//L2G2
arrfbLysGruppe[2]( 
	nZoneID:= 1, 
	bButtonZone1:= bTopButtonZone1,
	bBottomButtonZone1 := bBottomButtonZone1,
	//bButtonZone2:= bButtonZone2,
	fLuxOn:= fLuxOn, 
	fLuxDim:= fLuxDim, 
	tPIRDim:= tPIRDim, 
	tPIROff:= tPIROff, 
	fOffsetSec:= fOffsetSec, 
	bReInit:= , 
	stDaliSetup:= arrstDaliSetupGruppe[2], 
	ipCommunication_Prim:= P_DALI_Background.arrfbKL6821Communication[arrDALI_LINE_NUM_LIGHT[2]], 
	//ipCommunication_Sec:= P_DALI_Background.arrfbKL6821Communication[arrDALI_LINE_NUM_LIGHT[2]], 
	//ipCommunication_Supl:= P_DALI_Background.arrfbKL6821Communication[arrDALI_LINE_NUM_PENDANTS[2]], 
	fMinOutputPowerLevelRoom:= 15, 
	fMaxOutputPowerLevelRoom:= 100, 
	nCycleTimeInMS:= SH_Light.DALI_Param.nPlcTaskCycleTimeInMS*nDimCmdCycleTimeFactor,  //Used only for dim. Factor=2 makes dimming smooth 
	bRunTuning:= arrRunTuningGruppe[2], 
	bOccupiedRoom=> , 
	bError_Prim=> , 
	nError_Prim=> , 
	stTuneData:=arrstTuneDataGruppe[2] , 
	stPirSensorData:= stPirSensorData, 					//samme sensordata
	stLiveData:= arrstLiveDataGruppe[2]);
END_ACTION

ACTION A_ModbusComm:
//Manage data for modbus communication

//Manage data for read-only in PLC
stRoomDataPLC.bPirActive			:= stPirSensorData.bPrc;
stRoomDataPLC.uiActLuxLevel			:= TO_UINT(TRUNC(stPirSensorData.fBrightness));
stRoomDataPLC.uiActLightLevelPct	:= TO_UINT(TRUNC(arrfbLysGruppe[1].fbBallast.fActlLgtLvl_Prim));
		//stRoomDataPLC.uiActLightLevelPct	:= TO_UINT(TRUNC(fbLys.fbBallast.fActlLgtLvl_Prim)); //if only one group light control
stRoomDataPLC.uiBallastOnHours		:= uiBallastOnHours_MB; //The calculation for BallastOnHours is stored directly to the MB register below


//Assign data for read-only to MB registers
bPirActive_MB		:= stRoomDataPLC.bPirActive;
uiActLuxLevel_MB	:= stRoomDataPLC.uiActLuxLevel;

	//calculate BallastOnHours
	fbBallastOnHours(
		bEnableHourCount	:= bEnableHourCount,
		bPauseCount			:= arrfbLysGruppe[1].fbLightCtrl.bOffZone1,
		uiOnHours			:= uiBallastOnHours_MB,			//OnHours is updated here
		byOverflowCount		:= byOnHoursOverflowCount);


//Manage data for read/write for both PLC and MB registers
fbWriteSPLuxLevel(	nMaxValOut	:= uiMaxLuxLevel,
					nValIn1		:= uiSPLuxLevel_MB,		//nValIn1 takes priotity in case of download or restart
					nValIn2		:= stRoomDataPLC.uiSpLuxLevel,
					nValOut		=> uiLuxOn
				);


fbWritePirDelayTIme(	nMaxValOut	:= uiMaxPirOffMinutes,
						nValIn1		:= uiPirOffDelayTime_MB,		//nValIn1 takes priotity in case of download or restart
						nValIn2		:= stRoomDataPLC.uiPirOffDelayTime,
						nValOut		=> uiPirOffMinutes
					);
					

//Convert read/write modbus data to appropriate datatypes in PLC
fLuxOn	:= TO_REAL(uiLuxOn);			
tPIROff	:= TO_TIME(uiPirOffMinutes*udTimeScaling); //Time conversion defaults to ms

fLuxDim	:= TO_REAL(stRoomDataPLC.uiSpDimLuxLevel);			
tPIRDim	:= TO_TIME(stRoomDataPLC.uiPirDimDelayTime*udTimeScaling); //Time conversion defaults to ms
END_ACTION

ACTION A_Sensor:

fbSensor.ipCommunication := P_DALI_Background.arrfbKL6821Communication[Sensor_DALI_LINE_NUM];

//only 1 sensor
fbSensor(
	byShrtAdr:= bySensorAddr,
	bInitialize:= bInitialize, 
	DALI_LINE_NUM:= Sensor_DALI_LINE_NUM, 
 	//bCancelHoldTimerOccupancy:= bCancelHoldTimerOccupancy, 
	stSensorSetup := stDaliSensorSetup,
	bInitErr=> bInitErr, 
	bInitDone=> bInitDone,
	stPirSensorData:= stPirSensorData, 
	arrSensorScales:= arrSensorScales);


//several sensors
(*	
fbSensor(
	arrShrtAdr:= arrSensorAddr,
	bInitialize:= bInitialize, 
	DALI_LINE_NUM:= Sensor_DALI_LINE_NUM, 
 	//bCancelHoldTimerOccupancy:= bCancelHoldTimerOccupancy, 
	stSensorSetup := stDaliSensorSetup,
	arrInitErr=> arrInitErr, 
	arrInitDone=> arrInitDone,
	stPirSensorData:= stPirSensorData, 
	arrSensorScales:= arrSensorScales);
	*)
END_ACTION

END_PROGRAM

// ---- POUs/Alle_Rum/Rum_Med_DALI_Pir/Rum_4_213_Og_4_215_Foldedoer/P_Rum_4_215.TcPOU
PROGRAM P_Rum_4_215
VAR
(*Rummet består af to lysgrupper - L1G7 og L2G7 - på to forskellige linjer
Begge grupper afhænger af samme PIR-input - pir-adr. 5 og 8 - på DALI-linje 2.
Derfor oprettes to adskilte reguleringer med samme PV.
Yderligere logik for knapfunktion og pirsignaler håndteres i program for foldedør.
*)

	arrfbLysGruppe			: ARRAY [1..2] OF SH_Light.FB_Light_Type_A;
	arrstDaliSetupGruppe	: ARRAY [1..2] OF SH_Light.ST_DALI_RoomSetup := 
	
													[(	byShrtAdr_Prim := 18, 
														byGrpAdr_Prim := 7, 
														eMod_Prim := E_DALIAddressType.Group, 
														//byShrtAdr_Sec := 1, 
														//byGrpAdr_Sec := 1, 
														//eMod_Sec := E_DALIAddressType.Short, 
														//byShrtAdr_Supl := 1,
														//byGrpAdr_Supl := 1,
														//eMod_Supl := E_DALIADDRESSTYPE.Group,
														DALI_LINE_NUM_PRIM := arrDALI_LINE_NUM_LIGHT[1], 
														DALI_LINE_NUM_SEC := 0, //0 = ingen zonestyring/vinduerække
														DALI_LINE_NUM_SUPL := arrDALI_LINE_NUM_PENDANTS[1]),
														
													(	byShrtAdr_Prim := 13, 
														byGrpAdr_Prim := 7, 
														eMod_Prim := E_DALIAddressType.Group,
														//byShrtAdr_Sec := 1, 
														//byGrpAdr_Sec := 1, 
														//eMod_Sec := E_DALIAddressType.Short, 
														//byShrtAdr_Supl := 1,
														//byGrpAdr_Supl := 1,
														//eMod_Supl := E_DALIAddressType.Group, 
														DALI_LINE_NUM_PRIM := arrDALI_LINE_NUM_LIGHT[2], 
														DALI_LINE_NUM_SEC := 0, 
														DALI_LINE_NUM_SUPL := arrDALI_LINE_NUM_PENDANTS[2])];
														
	arrstLiveDataGruppe		: ARRAY [1..2] OF SH_Light.ST_LiveData;
	
	arrRunTuningGruppe: ARRAY[1..2] OF BOOL;
	
	bTopButtonZone1				: BOOL;
	bTopButtonZone1_Visu		: BOOL;
	bBottomButtonZone1			: BOOL;
	bBottomButtonZone1_Visu	: BOOL;
	bButtonZone2					: BOOL;
	bNeighborRoomsPir			: BOOL;
	fLuxOn								: REAL; 
	fLuxDim							: REAL;
	tPIRDim							: TIME;
	tPIROff							: TIME;
	fOffsetSec						: REAL := 20;
 

// Sensor Settings
	//fbSensor					: SH_Light.FB_NIKO_P46xx_1Pcs;
	fbSensor						: SH_Light.FB_NIKO_P46xx_2Pcs;
	//bySensorAddr				: BYTE := 1;
	arrSensorAddr				: ARRAY[1..2] OF BYTE := [5,8];
	bInitialize						: BOOL := TRUE;
	stDaliSensorSetup			: ST_DALI_NIKOP46SetupData;
	//bInitErr							: BOOL;
	//bInitDone						: BOOL;
	arrInitErr						: ARRAY [1..2] OF BOOL;
	arrInitDone					: ARRAY [1..2] OF BOOL;
	arrSensorScales				: ARRAY [1..10] OF SH_Light.ST_DALI_SensorScaleMode :=
																					[	(fMeassureMaxSensor := rMeassure_Zone5, fReadMaxSensor := rRead_Zone5),																		
																						(fMeassureMaxSensor := rMeassure_Zone5, fReadMaxSensor := rRead_Zone5),	
																						8(())];
																																			
	bCancelHoldTimerOccupancy	: BOOL;
(*	eEventPriorityOccupancy		: E_DALIEventPriority := E_DALIEVENTPRIORITY.Middle;
	nHoldTimerOccupancy			: WORD := 5; // Value in s. 	
	nReportTimerOccupancy		: BYTE := 120; // Value in s, Preset manufacturer value
	nDeadtimeTimerOccupancy		: WORD := 100; // Value in ms, Predefined Value of DALI Standard
	bCancelHoldTimerOccupancy	: BOOL;
	nSensitivityOccupancy		: BYTE:= 3; //setting Sensivity (0..4) 0 (Off), 1 (Min), 2(Low), 3(High) and 4 (Max)

	bEnableLuxEvent				: BOOL;
	eEventPriorityBrightness	: E_DALIEventPriority := E_DALIEVENTPRIORITY.Middle;
	nDeadtimeTimerBrightness	: WORD := 1500; // Value in ms, Predefined Value of DALI Standard
	nHysteresisBrightness		: BYTE := 2; // Value in %
	nHysteresisMinBrightness	: BYTE := 10; // Absolute Value, depending on the manufacturer specific resolution
	nReportTimerBrightness		: BYTE := 120; // Value in s, Preset manufacturer value
*)


//ModbusComm setup
	
	fbWriteSPLuxLevel				: SH_Light.FB_TwoVal_SelectOne_RTrigChange;
	fbWritePirDelayTIme			: SH_Light.FB_TwoVal_SelectOne_RTrigChange;
	stRoomDataPLC					: SH_Light.ST_RoomDataPLC	:=	(	uiPirOffDelayTime	:= 30,
																										uiSpLuxLevel			:= 500,
																										uiPirDimDelayTime	:= 15,
																										uiSpDimLuxLevel		:= 200);
																
	fbBallastOnHours					: SH_Light.FB_CountOnHours;
	bEnableHourCount				: BOOL := TRUE;
	
	//Non-persistent modbus data
	bPirActive_MB					AT%MX144.0	: BOOL;				//bPirLys i gammel kode
	uiActLuxLevel_MB			AT%MB148		: UINT;				//intHMIAktueltLux i gammel kode
	uiActLightLevelPct_MB	AT%MB156		: UINT;				//intDALI_Gruppe1_Lysniveau i gammel kode
	
	//For Conversion
	uiPirOffMinutes						: UINT;
	udTimeScaling						: UDINT := 60000;
	uiLuxOn								: UINT;
	
	//max values checks
	uiMaxLuxLevel						: UINT := 1023;
	uiMaxPirOffMinutes					: UINT := 180;
	
END_VAR

VAR CONSTANT
	Sensor_DALI_LINE_NUM					: BYTE := 2;
	arrDALI_LINE_NUM_LIGHT				: ARRAY[1..2] OF BYTE := [1,2]; //korrekt rækkefølge nødvendig //rækkefølge og linje 
	arrDALI_LINE_NUM_PENDANTS	: ARRAY[1..2] OF BYTE := [0,0]; //korrekt rækkefølge nødvendig. 0 = ingen pendler
END_VAR

VAR PERSISTENT
	stPirSensorData										: SH_Light.ST_DALI_Sensor;
	arrstTuneDataGruppe								: ARRAY [1..2] OF SH_Light.ST_TuneData_EX;

	uiPirOffDelayTime_MB		AT%MB146	    : UINT;				//intHMI_Pir_SetValue i gammel kode
	uiSPLuxLevel_MB		    AT%MB152    	: UINT;				//intHMI_Lux_SetValue i gammel kode
	uiBallastOnHours_MB	    AT%MB158	    : UINT;				//dintHMILysbraendtimer1 i gammel kode
	byOnHoursOverflowCount			   				: BYTE;
END_VAR

A_Buttons();
A_LightCtrl();
A_ModbusComm();
A_Sensor();

ACTION A_Buttons:
//Logik for knapper håndteres i P_Foldedoer_4_213

bTopButtonZone1		:= P_Foldedoer_4_213.arrTopButtonZone1Comb[2] OR bTopButtonZone1_Visu;
bBottomButtonZone1	:= P_Foldedoer_4_213.arrBottomButtonZone1Comb[2] OR bBottomButtonZone1_Visu;
END_ACTION

ACTION A_LightCtrl:
  
//gruppe L1G1
arrfbLysGruppe[1]( 
	nZoneID:= 1, 
	bButtonZone1:= bTopButtonZone1,
	bBottomButtonZone1 := bBottomButtonZone1,
	//bButtonZone2:= bButtonZone2,
	fLuxOn:= fLuxOn, 
	fLuxDim:= fLuxDim, 
	tPIRDim:= tPIRDim, 
	tPIROff:= tPIROff, 
	fOffsetSec:= fOffsetSec, 
	bReInit:= , 
	stDaliSetup:= arrstDaliSetupGruppe[1], 
	ipCommunication_Prim:= P_DALI_Background.arrfbKL6821Communication[arrDALI_LINE_NUM_LIGHT[1]], 
	//ipCommunication_Sec:= P_DALI_Background.arrfbKL6821Communication[arrDALI_LINE_NUM_LIGHT[1]], 
	//ipCommunication_Supl:= P_DALI_Background.arrfbKL6821Communication[arrDALI_LINE_NUM_PENDANTS[1]], 
	fMinOutputPowerLevelRoom:= 15, 
	fMaxOutputPowerLevelRoom:= 100, 
	nCycleTimeInMS:= SH_Light.DALI_Param.nPlcTaskCycleTimeInMS*nDimCmdCycleTimeFactor,   //Used only for dim. Factor=2 makes dimming smooth
	bRunTuning:= arrRunTuningGruppe[1], 
	bOccupiedRoom=> , 
	bError_Prim=> , 
	nError_Prim=> , 
	stTuneData:=arrstTuneDataGruppe[1] , 
	stPirSensorData:=  P_Foldedoer_4_213.arrstPirSensorDataComb[2], 					//samme sensordata
	stLiveData:= arrstLiveDataGruppe[1]);

//gruppe 15	
arrfbLysGruppe[2]( 
	nZoneID:= 1, 
	bButtonZone1:= bTopButtonZone1,
	bBottomButtonZone1 := bBottomButtonZone1,
	//bButtonZone2:= bButtonZone2,
	fLuxOn:= fLuxOn, 
	fLuxDim:= fLuxDim, 
	tPIRDim:= tPIRDim, 
	tPIROff:= tPIROff, 
	fOffsetSec:= fOffsetSec, 
	bReInit:= , 
	stDaliSetup:= arrstDaliSetupGruppe[2], 
	ipCommunication_Prim:= P_DALI_Background.arrfbKL6821Communication[arrDALI_LINE_NUM_LIGHT[2]], 
	//ipCommunication_Sec:= P_DALI_Background.arrfbKL6821Communication[arrDALI_LINE_NUM_LIGHT[2]], 
	//ipCommunication_Supl:= P_DALI_Background.arrfbKL6821Communication[arrDALI_LINE_NUM_PENDANTS[2]], 
	fMinOutputPowerLevelRoom:= 15, 
	fMaxOutputPowerLevelRoom:= 100, 
	nCycleTimeInMS:= SH_Light.DALI_Param.nPlcTaskCycleTimeInMS*nDimCmdCycleTimeFactor,  //Used only for dim. Factor=2 makes dimming smooth
	bRunTuning:= arrRunTuningGruppe[2], 
	bOccupiedRoom=> , 
	bError_Prim=> , 
	nError_Prim=> , 
	stTuneData:=arrstTuneDataGruppe[2] , 
	stPirSensorData:=  P_Foldedoer_4_213.arrstPirSensorDataComb[2], 					//samme sensordata
	stLiveData:= arrstLiveDataGruppe[2]);
END_ACTION

ACTION A_ModbusComm:
//Manage data for modbus communication

//Manage data for read-only in PLC
stRoomDataPLC.bPirActive			:= stPirSensorData.bPrc;
stRoomDataPLC.uiActLuxLevel			:= TO_UINT(TRUNC(stPirSensorData.fBrightness));
stRoomDataPLC.uiActLightLevelPct	:= TO_UINT(TRUNC(arrfbLysGruppe[1].fbBallast.fActlLgtLvl_Prim));
		//stRoomDataPLC.uiActLightLevelPct	:= TO_UINT(TRUNC(fbLys.fbBallast.fActlLgtLvl_Prim)); //if only one group light control
stRoomDataPLC.uiBallastOnHours		:= uiBallastOnHours_MB; //The calculation for BallastOnHours is stored directly to the MB register below


//Assign data for read-only to MB registers
bPirActive_MB		:= stRoomDataPLC.bPirActive;
uiActLuxLevel_MB	:= stRoomDataPLC.uiActLuxLevel;

	//calculate BallastOnHours
	fbBallastOnHours(
		bEnableHourCount	:= bEnableHourCount,
		bPauseCount			:= arrfbLysGruppe[1].fbLightCtrl.bOffZone1,
		uiOnHours			:= uiBallastOnHours_MB,			//OnHours is updated here
		byOverflowCount		:= byOnHoursOverflowCount);


//Manage data for read/write for both PLC and MB registers
fbWriteSPLuxLevel(	nMaxValOut	:= uiMaxLuxLevel,
					nValIn1		:= uiSPLuxLevel_MB,		//nValIn1 takes priotity in case of download or restart
					nValIn2		:= stRoomDataPLC.uiSpLuxLevel,
					nValOut		=> uiLuxOn
				);


fbWritePirDelayTIme(	nMaxValOut	:= uiMaxPirOffMinutes,
						nValIn1		:= uiPirOffDelayTime_MB,		//nValIn1 takes priotity in case of download or restart
						nValIn2		:= stRoomDataPLC.uiPirOffDelayTime,
						nValOut		=> uiPirOffMinutes
					);
					

//Convert read/write modbus data to appropriate datatypes in PLC
fLuxOn	:= TO_REAL(uiLuxOn);			
tPIROff	:= TO_TIME(uiPirOffMinutes*udTimeScaling); //Time conversion defaults to ms

fLuxDim	:= TO_REAL(stRoomDataPLC.uiSpDimLuxLevel);			
tPIRDim	:= TO_TIME(stRoomDataPLC.uiPirDimDelayTime*udTimeScaling); //Time conversion defaults to ms
END_ACTION

ACTION A_Sensor:

fbSensor.ipCommunication := P_DALI_Background.arrfbKL6821Communication[Sensor_DALI_LINE_NUM];

//only 1 sensor
(*
fbSensor(
	byShrtAdr:= bySensorAddr,
	bInitialize:= bInitialize, 
	DALI_LINE_NUM:= Sensor_DALI_LINE_NUM, 
 	//bCancelHoldTimerOccupancy:= bCancelHoldTimerOccupancy, 
	stSensorSetup := stDaliSensorSetup,
	bInitErr=> bInitErr, 
	bInitDone=> bInitDone,
	stPirSensorData:= stPirSensorData, 
	arrSensorScales:= arrSensorScales);
*)

//several sensors
fbSensor(
	arrShrtAdr:= arrSensorAddr,
	bInitialize:= bInitialize, 
	DALI_LINE_NUM:= Sensor_DALI_LINE_NUM, 
 	//bCancelHoldTimerOccupancy:= bCancelHoldTimerOccupancy, 
	stSensorSetup := stDaliSensorSetup,
	arrInitErr=> arrInitErr, 
	arrInitDone=> arrInitDone,
	stPirSensorData := P_Foldedoer_4_213.arrstPirSensorData[2], 
	arrSensorScales:= arrSensorScales);
	
	stPirSensorData := P_Foldedoer_4_213.arrstPirSensorData[2]; //For at holde samme navngivning i A_ModbusComm
END_ACTION

END_PROGRAM

// ---- POUs/Alle_Rum/Gange/Gang_4_210A/P_Gang_4_210A.TcPOU
PROGRAM P_Gang_4_210A
VAR
//Light

	fbLys			: SH_Light.FB_Light_Type_B;
	
	stDaliSetup	: SH_Light.ST_DALI_RoomSetup := (
														byShrtAdr_Prim	:= 56, 
														byGrpAdr_Prim		:= 1, 
														eMod_Prim			:= E_DALIAddressType.Group, 
														//byShrtAdr_Sec	:= 1, 
														//byGrpAdr_Sec	:= 1, 
														//eMod_Sec			:= E_DALIAddressType.Short, 
														//byShrtAdr_Supl		:= 1,
														//byGrpAdr_Supl		:= 1,
														//eMod_Supl			:= Tc3_DALI.E_DALIAddressType.Short, 
														DALI_LINE_NUM_PRIM := DALI_LINE_NUM_LIGHT, 
														DALI_LINE_NUM_SEC := 0, 
														DALI_LINE_NUM_SUPL := DALI_LINE_NUM_PENDANT);
														
	stLiveData						: SH_Light.ST_LiveData;
	bRunTuning						: BOOL;
	
	bTopButtonZone1				: BOOL;
	bTopButtonZone1_Visu		: BOOL;
	bBottomButtonZone1			: BOOL;
	bBottomButtonZone1_Visu	: BOOL;
	bButtonZone2					: BOOL;
	fLuxOn								: REAL;
	fLuxDim							: REAL;
	tPIRDim							: TIME;
	tPIROff							: TIME;
	fOffsetSec						: REAL := 20;
	bOccupiedRoom				: BOOL;
	
// Sensor Settings
	fbSensor							: SH_Light.FB_NIKO_P46xx_1Pcs;
	//fbSensor							: SH_Light.FB_NIKO_P46xx_2Pcs;
	bySensorAddr					: BYTE := 63;
	//arrSensorAddr					: ARRAY[1..2] OF BYTE := [3,4];
	bInitialize							: BOOL := TRUE;
	stDaliSensorSetup				: ST_DALI_NIKOP46SetupData;
	bInitErr								: BOOL;
	bInitDone							: BOOL;
	//arrInitErr							: ARRAY [1..2] OF BOOL;
	//arrInitDone						: ARRAY [1..2] OF BOOL;
	arrSensorScales					: ARRAY [1..10] OF SH_Light.ST_DALI_SensorScaleMode :=
																						[	(fMeassureMaxSensor := rMeassure_Zone10, fReadMaxSensor := rRead_Zone10),
																							9(())];
	bCancelHoldTimerOccupancy	: BOOL;
(*	eEventPriorityOccupancy		: E_DALIEventPriority := E_DALIEVENTPRIORITY.Middle;
	nHoldTimerOccupancy			: WORD := 5; // Value in s. 	
	nReportTimerOccupancy		: BYTE := 120; // Value in s, Preset manufacturer value
	nDeadtimeTimerOccupancy		: WORD := 100; // Value in ms, Predefined Value of DALI Standard
	bCancelHoldTimerOccupancy	: BOOL;
	nSensitivityOccupancy		: BYTE:= 3; //setting Sensivity (0..4) 0 (Off), 1 (Min), 2(Low), 3(High) and 4 (Max)

	bEnableLuxEvent				: BOOL;
	eEventPriorityBrightness	: E_DALIEventPriority := E_DALIEVENTPRIORITY.Middle;
	nDeadtimeTimerBrightness	: WORD := 1500; // Value in ms, Predefined Value of DALI Standard
	nHysteresisBrightness		: BYTE := 2; // Value in %
	nHysteresisMinBrightness	: BYTE := 10; // Absolute Value, depending on the manufacturer specific resolution
	nReportTimerBrightness		: BYTE := 120; // Value in s, Preset manufacturer value
*)

//ModbusComm setup
	
	fbWriteSPLuxLevel				: SH_Light.FB_TwoVal_SelectOne_RTrigChange;
	fbWritePirDelayTIme			: SH_Light.FB_TwoVal_SelectOne_RTrigChange;
	stRoomDataPLC					: SH_Light.ST_RoomDataPLC	:=	(	uiPirOffDelayTime	:= 30,
																										uiSpLuxLevel			:= 500,
																										uiPirDimDelayTime	:= 15,
																										uiSpDimLuxLevel		:= 200);
																
	fbBallastOnHours					: SH_Light.FB_CountOnHours;
	bEnableHourCount				: BOOL := TRUE;
	
	//Non-persistent modbus data
	bPirActive_MB					AT%MX200.0	: BOOL;				//bPirLys i gammel kode
	uiActLuxLevel_MB			AT%MB204		: UINT;				//intHMIAktueltLux i gammel kode
	uiActLightLevelPct_MB	AT%MB208		: UINT;				//intDALI_Gruppe1_Lysniveau i gammel kode
	
	//For Conversion
	uiPirOffMinutes						: UINT;
	udTimeScaling						: UDINT := 60000;
	uiLuxOn								: UINT;
	
	//max values checks
	uiMaxLuxLevel						: UINT := 1023;
	uiMaxPirOffMinutes				: UINT := 180;

END_VAR

VAR CONSTANT
	Sensor_DALI_LINE_NUM: BYTE := 3;
	DALI_LINE_NUM_LIGHT: BYTE := 3;
	DALI_LINE_NUM_PENDANT: BYTE :=0;
END_VAR
VAR PERSISTENT
	stPirSensorData: SH_Light.ST_DALI_Sensor;
	stTuneData: SH_Light.ST_TuneData_EX;
	
	uiPirOffDelayTime_MB		AT%MB202	    : UINT;				//intHMI_Pir_SetValue i gammel kode
	uiSPLuxLevel_MB		    AT%MB206    	: UINT;				//intHMI_Lux_SetValue i gammel kode
	uiBallastOnHours_MB	    AT%MB210	    : UINT;				//dintHMILysbraendtimer1 i gammel kode
	byOnHoursOverflowCount			   				: BYTE;
END_VAR

A_Buttons();
A_LightCtrl();
A_ModbusComm();
A_Sensor();

ACTION A_Buttons:
bTopButtonZone1		:= 	bTopButtonZone1_Visu;
bBottomButtonZone1	:= 	bBottomButtonZone1_Visu;
END_ACTION

ACTION A_LightCtrl:

fbLys(
	nZoneID:= 1, 
	bButtonZone1:= bTopButtonZone1,
	bBottomButtonZone1 := bBottomButtonZone1, 
	//bButtonZone2:= bButtonZone2, 
	fLuxOn:= fLuxOn, 
	fLuxDim:= fLuxDim, 
	tPIRDim:= tPIRDim, 
	tPIROff:= tPIROff, 
	fOffsetSec:= fOffsetSec, 
	bReInit:= , 
	stDaliSetup:= stDaliSetup, 
	ipCommunication_Prim:= P_DALI_Background.arrfbKL6821Communication[DALI_LINE_NUM_LIGHT], 
	//ipCommunication_Sec:= P_DALI_Background.arrfbKL6821Communication[DALI_LINE_NUM_LIGHT], 
	//ipCommunication_Supl:= P_DALI_Background.arrfbKL6821Communication[DALI_LINE_NUM_PENDANT],
	fMinOutputPowerLevelRoom:= 15, 
	fMaxOutputPowerLevelRoom:= 100, 
	nCycleTimeInMS:= SH_Light.DALI_Param.nPlcTaskCycleTimeInMS*nDimCmdCycleTimeFactor,  //Used only for dim. Factor=2 makes dimming smooth
	bRunTuning:= bRunTuning, 
	bOccupiedRoom=> bOccupiedRoom, 
	bError_Prim=> , 
	nError_Prim=> , 
	stTuneData:=stTuneData , 
	stPirSensorData:= stPirSensorData, 
	stLiveData:= stLiveData);
END_ACTION

ACTION A_ModbusComm:
//Manage data for modbus communication

//Manage data for read-only in PLC
stRoomDataPLC.bPirActive			:= stPirSensorData.bPrc;
stRoomDataPLC.uiActLuxLevel			:= TO_UINT(TRUNC(stPirSensorData.fBrightness));
stRoomDataPLC.uiActLightLevelPct	:= TO_UINT(TRUNC(fblys.fbBallast.fActlLgtLvl_Prim));
		//stRoomDataPLC.uiActLightLevelPct	:= TO_UINT(TRUNC(fbLys.fbBallast.fActlLgtLvl_Prim)); //if only one group light control
stRoomDataPLC.uiBallastOnHours		:= uiBallastOnHours_MB; //The calculation for BallastOnHours is stored directly to the MB register below


//Assign data for read-only to MB registers
bPirActive_MB		:= stRoomDataPLC.bPirActive;
uiActLuxLevel_MB	:= stRoomDataPLC.uiActLuxLevel;

	//calculate BallastOnHours
	fbBallastOnHours(
		bEnableHourCount	:= bEnableHourCount,
		bPauseCount			:= fbLys.fbLightCtrl.bOffZone1,
		uiOnHours			:= uiBallastOnHours_MB,			//OnHours is updated here
		byOverflowCount		:= byOnHoursOverflowCount);


//Manage data for read/write for both PLC and MB registers
fbWriteSPLuxLevel(	nMaxValOut	:= uiMaxLuxLevel,
					nValIn1		:= uiSPLuxLevel_MB,		//nValIn1 takes priotity in case of download or restart
					nValIn2		:= stRoomDataPLC.uiSpLuxLevel,
					nValOut		=> uiLuxOn
				);


fbWritePirDelayTIme(	nMaxValOut	:= uiMaxPirOffMinutes,
						nValIn1		:= uiPirOffDelayTime_MB,		//nValIn1 takes priotity in case of download or restart
						nValIn2		:= stRoomDataPLC.uiPirOffDelayTime,
						nValOut		=> uiPirOffMinutes
					);
					

//Convert read/write modbus data to appropriate datatypes in PLC
fLuxOn	:= TO_REAL(uiLuxOn);			
tPIROff	:= TO_TIME(uiPirOffMinutes*udTimeScaling); //Time conversion defaults to ms

fLuxDim	:= TO_REAL(stRoomDataPLC.uiSpDimLuxLevel);			
tPIRDim	:= TO_TIME(stRoomDataPLC.uiPirDimDelayTime*udTimeScaling); //Time conversion defaults to ms
END_ACTION

ACTION A_Sensor:

fbSensor.ipCommunication := P_DALI_Background.arrfbKL6821Communication[Sensor_DALI_LINE_NUM];


fbSensor(
	byShrtAdr:= bySensorAddr,
	bInitialize:= bInitialize, 
	DALI_LINE_NUM:= Sensor_DALI_LINE_NUM, 
 	//bCancelHoldTimerOccupancy:= bCancelHoldTimerOccupancy, 
	stSensorSetup := stDaliSensorSetup,
	bInitErr=> bInitErr, 
	bInitDone=> bInitDone,
	stPirSensorData:= stPirSensorData, 
	arrSensorScales:= arrSensorScales);


(*
fbSensor(
	arrShrtAdr:= arrSensorAddr,
	bInitialize:= bInitialize, 
	DALI_LINE_NUM:= Sensor_DALI_LINE_NUM, 
 	//bCancelHoldTimerOccupancy:= bCancelHoldTimerOccupancy, 
	stSensorSetup := stDaliSensorSetup,
	arrInitErr=> arrInitErr, 
	arrInitDone=> arrInitDone,
	stPirSensorData:= stPirSensorData, 
	arrSensorScales:= arrSensorScales);
	*)
END_ACTION

END_PROGRAM

// ---- POUs/Alle_Rum/Trapper/P_DigTest.TcPOU
PROGRAM P_DigTest
VAR
	DigIn1		AT %I*	: BOOL;
	DigIn2						: BOOL;
	DigIn3		AT %I*	: BOOL;
	DigIn4		AT %I*	: BOOL;
	DigIn5		AT %I*	: BOOL;
	DigIn6		AT %I*	: BOOL;
	DigIn7		AT %I*	: BOOL;
	DigIn8		AT %I*	: BOOL;
END_VAR

END_PROGRAM

// ---- POUs/EnOcean/P_EnOcean.TcPOU
PROGRAM P_EnOcean
VAR
	fbKL6581			: FB_KL6581;
	stKL6581_in  AT %I* : KL6581_INPUT;
	stKL6581_out AT %Q*	: KL6581_OUTPUT;
	stKL6581			: STR_KL6581;
	bInitCom			: BOOL := TRUE;
	
	arrEnOcean_Search	: ARRAY [1..8] OF FB_EnOcean_Search;
	nSearchIdx			: BYTE;
	bSerach				: BOOL;
	arrDevices			: ARRAY [1..8] OF INT;
	arrID				: ARRAY [1..8, 0..255] OF DWORD;
	
	//Trykknapper Atrium
	fbGang_3_109_Kantine_Tryk_PladeA	: FB_Rec_RPS_Switch;
	fbAtriumNiveau_Tryk_PladeB				: FB_Rec_RPS_Switch;
	fbAtriumNiveau_Tryk_Sevice				: FB_Rec_RPS_Switch;
	
	//Trykknapper på gange
	fbGang_4_211_Tryk_Indgang				: FB_Rec_RPS_Switch;
	fbGang_4_211_Tryk_Ekstra					: FB_Rec_RPS_Switch;
	
	//Trykknapper i rum
	fbRum_4_206_Tryk_Indgang					: FB_Rec_RPS_Switch;
	fbRum_4_206_Tryk_Ekstra					: FB_Rec_RPS_Switch;
	
	fbRum_4_207_Tryk_Indgang					: FB_Rec_RPS_Switch;
	fbRum_4_207_Tryk_Ekstra					: FB_Rec_RPS_Switch;
	
	fbRum_4_211A_Tryk_Indgang				: FB_Rec_RPS_Switch;
	fbRum_4_211A_Tryk_Ekstra					: FB_Rec_RPS_Switch;
	
	fbRum_4_213_Tryk_Indgang					: FB_Rec_RPS_Switch;
	fbRum_4_213_Tryk_Pendler					: FB_Rec_RPS_Switch;
	
	fbRum_4_215_Tryk								: FB_Rec_RPS_Switch;
	
END_VAR

VAR CONSTANT
	byNode_1: BYTE := 1;
	byNode_2: BYTE := 2;
	byNode_3: BYTE := 3;
	byNode_4: BYTE := 4;
	byNode_5: BYTE := 5;
	byNode_6: BYTE := 6;
	byNode_7: BYTE := 7;
	byNode_8: BYTE := 8;
END_VAR


(* Kommunikation mit der KL6581. *)
(* Communication with the KL6581. *)
fbKL6581(
	bInit			:= bInitCom,
	nIdx			:= 2,
	stKL6581_in		:= stKL6581_In,
	stKL6581_out	:= stKL6581_Out,
	bReady			=> ,
	bBusy			=> ,
	bError			=> ,
	iErrorID		=> ,
	str_KL6581		=> stKL6581);
	
GVL_AHDataModbus.EnOceanError	:= TO_UINT(fbKL6581.iErrorID);

(* Warten bis der Kommunikationsbaustein initialisiert wurde.*)
(* Wait until the communication function block has been initialized. *)
IF (NOT fbKL6581.bReady) THEN
	RETURN;
END_IF

FOR nSearchIdx:= 1 TO 8 DO
	arrEnOcean_Search[nSearchIdx](
		bStart:= TRUE, 
		str_KL6581:= stKL6581 , 
		byNode:= nSearchIdx, 
		bReceive=> , 
		iDevices=>arrDevices[nSearchIdx] , 
		ar_ID=> );
		
		MEMCPY(ADR(arrID[nSearchIdx,0]), ADR(arrEnOcean_Search[nSearchIdx].ar_ID), SIZEOF(arrEnOcean_Search[nSearchIdx].ar_ID)); 
END_FOR

//Atrium Niveauer
A_AtriumNiveau();

//Gange
A_Gang_1_309_Kantine();
A_Gang_4_211();

//Rum
A_Rum_4_206();
A_Rum_4_207();
A_Rum_4_211A();
A_Rum_4_213();
A_Rum_4_215();

ACTION A_AtriumNiveau:
fbAtriumNiveau_Tryk_PladeB(
	str_KL6581:=stKL6581 , 
	byNode:=0 , 
	dw_ID:= 16#0029B92D, 
	str_EnOceanSwitch=> GVL_EnOcean.strEnOceanSwitch_AtriumNiveau_PladeB,
	by_Node=> , 
	bReceive=> );
(*
fbAtriumNiveau_Tryk_Sevice(
	str_KL6581:=stKL6581 , 
	byNode:=0, 
	dw_ID:= 16#00FEE4FE87, 
	str_EnOceanSwitch=> GVL_EnOcean.strEnOceanSwitch_AtriumNiveau_Service, 
	by_Node=> , 
	bReceive=> );
	*)
END_ACTION

ACTION A_Gang_1_309_Kantine:
fbGang_3_109_Kantine_Tryk_PladeA(
	str_KL6581:=stKL6581 , 
	byNode:=0, 
	dw_ID:= 16#0029B976, 
	str_EnOceanSwitch=> GVL_EnOcean.strEnOceanSwitch_Gang_3_109_PladeA, 
	by_Node=> , 
	bReceive=> );
END_ACTION

ACTION A_Gang_4_211:
fbGang_4_211_Tryk_Indgang(
	str_KL6581:=stKL6581 , 
	byNode:=byNode_4 , 
	dw_ID:= 16#0029EDF3, 
	str_EnOceanSwitch=> GVL_EnOcean.strEnOceanSwitch_Gang_4_211_Indgang, 
	by_Node=> , 
	bReceive=> );
	
fbGang_4_211_Tryk_Ekstra(
	str_KL6581:=stKL6581 , 
	byNode:=byNode_4 , 
	dw_ID:= 16#0029AB75, 
	str_EnOceanSwitch=> GVL_EnOcean.strEnOceanSwitch_Gang_4_211_Ekstra, 
	by_Node=> , 
	bReceive=> );
END_ACTION

ACTION A_Rum_4_206:
fbRum_4_206_Tryk_Indgang(
	str_KL6581:=stKL6581 , 
	byNode:=byNode_4 , 
	dw_ID:= 16#002F29CA, 
	str_EnOceanSwitch=> GVL_EnOcean.strEnOceanSwitch_Rum_4_206_Indgang, 
	by_Node=> , 
	bReceive=> );
	
fbRum_4_206_Tryk_Ekstra(
	str_KL6581:=stKL6581 , 
	byNode:=byNode_4 , 
	dw_ID:= 16#00290ED4, 
	str_EnOceanSwitch=> GVL_EnOcean.strEnOceanSwitch_Rum_4_206_Ekstra, 
	by_Node=> , 
	bReceive=> );
END_ACTION

ACTION A_Rum_4_207:
fbRum_4_207_Tryk_Indgang(
	str_KL6581:=stKL6581 , 
	byNode:=byNode_4 , 
	dw_ID:= 16#0029AD3E, 
	str_EnOceanSwitch=> GVL_EnOcean.strEnOceanSwitch_Rum_4_207_Indgang, 
	by_Node=> , 
	bReceive=> );
	
	fbRum_4_207_Tryk_Ekstra(
	str_KL6581:=stKL6581 , 
	byNode:=byNode_4, 
	dw_ID:= 16#0029AD8A, 
	str_EnOceanSwitch=> GVL_EnOcean.strEnOceanSwitch_Rum_4_207_Ekstra, 
	by_Node=> , 
	bReceive=> );
END_ACTION

ACTION A_Rum_4_211A:
fbRum_4_211A_Tryk_Indgang(
	str_KL6581:=stKL6581 , 
	byNode:=byNode_4 , 
	dw_ID:= 16#0029AD5B, 
	str_EnOceanSwitch=> GVL_EnOcean.strEnOceanSwitch_Rum_4_211A_Indgang, 
	by_Node=> , 
	bReceive=> );
	
fbRum_4_211A_Tryk_Ekstra(
	str_KL6581:=stKL6581 , 
	byNode:=byNode_4 , 
	dw_ID:= 16#0029AD80, 
	str_EnOceanSwitch=> GVL_EnOcean.strEnOceanSwitch_Rum_4_211A_Ekstra, 
	by_Node=> , 
	bReceive=> );
END_ACTION

ACTION A_Rum_4_213:
fbRum_4_213_Tryk_Indgang(
	str_KL6581:=stKL6581 , 
	byNode:=byNode_4 , 
	dw_ID:= 16#0029AB5C, 
	str_EnOceanSwitch=> GVL_EnOcean.strEnOceanSwitch_Rum_4_213_Indgang, 
	by_Node=> , 
	bReceive=> );
	
fbRum_4_213_Tryk_Pendler(
	str_KL6581:=stKL6581 , 
	byNode:=byNode_4 , 
	dw_ID:= 16#FEE4ED20, 
	str_EnOceanSwitch=> GVL_EnOcean.strEnOceanSwitch_Rum_4_213_Pendler, 
	by_Node=> , 
	bReceive=> );
END_ACTION

ACTION A_Rum_4_215:
fbRum_4_215_Tryk(
	str_KL6581:=stKL6581 , 
	byNode:=byNode_4 , 
	dw_ID:= 16#0029AADE, 
	str_EnOceanSwitch=> GVL_EnOcean.strEnOceanSwitch_Rum_4_215, 
	by_Node=> , 
	bReceive=> );
END_ACTION

END_PROGRAM

// ---- POUs/MAIN.TcPOU
PROGRAM MAIN
VAR
	nAlive: INT;
	breset: BOOL;
	nDemoVariable : INT;
	nCX8200_State	AT %I*	: UINT;
END_VAR

VAR PERSISTENT
	nDemoVar_Persist: INT;
END_VAR

nAlive:= nAlive + 1;
GVL_AHDataModbus.nCX8200_State_MB := nCX8200_State;

P_SystemDK.M_nCyclic(bReset := breset );
P_DALI_DIAG();
DALI_Commissioning();

P_DALI_Energy_Line();

P_AHModbusComm();

//Gange
P_Gang_3_109_Kantine();
P_Gang_4_208();
P_Gang_4_210A();
P_Gang_4_211();

//Foldedøre
P_Foldedoer_4_213();

//Rum
P_Rum_4_206();
P_Rum_4_207();
P_Rum_4_211A();

P_Rum_4_213();
P_Rum_4_215();

P_DigTest();

//P_DALI_Energy_Firmware_Test();

END_PROGRAM

// ---- POUs/Alle_Rum/Gange/Gang_3_109/Visualization_4_308.TcVIS
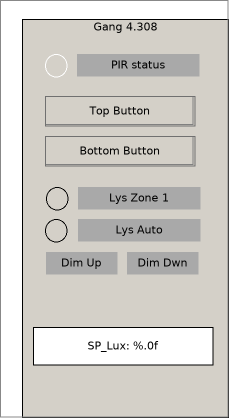
VISUALIZATION Visualization_4_308  // 229x418
    RoundedRectangle (22,19 207x399), "Gang 4.308"
    Rectangle (33,327 180x38), "SP_Lux: %.0f", text variable: P_Gang_3_109_Kantine.arrfbLysGruppe[1].fbLightCtrl.fLuxZone1
    Button (45,96 150x30), "Top Button"
        tap P_Gang_3_109_Kantine.bTopButtonZone1_Visu
    Button (45,136 150x30), "Bottom Button"
        tap P_Gang_3_109_Kantine.bBottomButtonZone1_Visu
    Ellipse (46,187 22x23), colour toggle: P_Gang_3_109_Kantine.arrfbLysGruppe[1].fbLightCtrl.bOnZone1
    Rectangle (78,187 122x22), "Lys Zone 1"
    Rectangle (46,252 71x22), "Dim Up", colour toggle: P_Gang_3_109_Kantine.arrfbLysGruppe[1].fbLightCtrl.bDimUp
    Rectangle (127,252 71x22), "Dim Dwn", colour toggle: P_Gang_3_109_Kantine.arrfbLysGruppe[1].fbLightCtrl.bDimDwn
    Ellipse (45,219 22x23), colour toggle: P_Gang_3_109_Kantine.arrfbLysGruppe[1].fbLightCtrl.bAutoZone1
    Rectangle (78,219 122x22), "Lys Auto"
    Ellipse (45,54 22x23), colour toggle: P_Gang_3_109_Kantine.arrfbLysGruppe[1].fbLightCtrl.bPIR
    Rectangle (77,54 122x22), "PIR status"
END_VISUALIZATION

// ---- POUs/Alle_Rum/Gange/Gang_4_208/Visualization_5_338_1.TcVIS
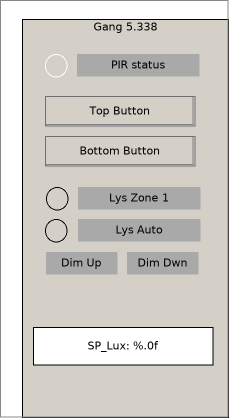
VISUALIZATION Visualization_5_338_1  // 229x418
    RoundedRectangle (22,19 207x399), "Gang 5.338"
    Rectangle (33,327 180x38), "SP_Lux: %.0f", text variable: P_Gang_5_338.arrfbLysGruppe[1].fbLightCtrl.fLuxZone1
    Button (45,96 150x30), "Top Button"
        tap P_Gang_5_338.bTopButtonZone1_Visu
    Button (45,136 150x30), "Bottom Button"
        tap P_Gang_5_338.bBottomButtonZone1_Visu
    Ellipse (46,187 22x23), colour toggle: P_Gang_5_338.arrfbLysGruppe[1].fbLightCtrl.bOnZone1
    Rectangle (78,187 122x22), "Lys Zone 1"
    Rectangle (46,252 71x22), "Dim Up", colour toggle: P_Gang_5_338.arrfbLysGruppe[1].fbLightCtrl.bDimUp
    Rectangle (127,252 71x22), "Dim Dwn", colour toggle: P_Gang_5_338.arrfbLysGruppe[1].fbLightCtrl.bDimDwn
    Ellipse (45,219 22x23), colour toggle: P_Gang_5_338.arrfbLysGruppe[1].fbLightCtrl.bAutoZone1
    Rectangle (78,219 122x22), "Lys Auto"
    Ellipse (45,54 22x23), colour toggle: P_Gang_5_338.arrfbLysGruppe[1].fbLightCtrl.bPIR
    Rectangle (77,54 122x22), "PIR status"
END_VISUALIZATION

// ---- POUs/Alle_Rum/Gange/Gang_4_211/Visualization_5_338_1_1_1_1.TcVIS
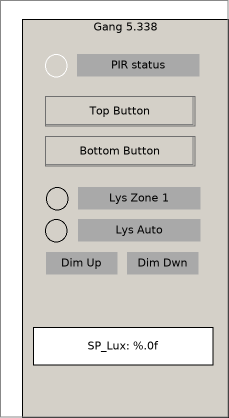
VISUALIZATION Visualization_5_338_1_1_1_1  // 229x418
    RoundedRectangle (22,19 207x399), "Gang 5.338"
    Rectangle (33,327 180x38), "SP_Lux: %.0f", text variable: P_Gang_5_338.arrfbLysGruppe[1].fbLightCtrl.fLuxZone1
    Button (45,96 150x30), "Top Button"
        tap P_Gang_5_338.bTopButtonZone1_Visu
    Button (45,136 150x30), "Bottom Button"
        tap P_Gang_5_338.bBottomButtonZone1_Visu
    Ellipse (46,187 22x23), colour toggle: P_Gang_5_338.arrfbLysGruppe[1].fbLightCtrl.bOnZone1
    Rectangle (78,187 122x22), "Lys Zone 1"
    Rectangle (46,252 71x22), "Dim Up", colour toggle: P_Gang_5_338.arrfbLysGruppe[1].fbLightCtrl.bDimUp
    Rectangle (127,252 71x22), "Dim Dwn", colour toggle: P_Gang_5_338.arrfbLysGruppe[1].fbLightCtrl.bDimDwn
    Ellipse (45,219 22x23), colour toggle: P_Gang_5_338.arrfbLysGruppe[1].fbLightCtrl.bAutoZone1
    Rectangle (78,219 122x22), "Lys Auto"
    Ellipse (45,54 22x23), colour toggle: P_Gang_5_338.arrfbLysGruppe[1].fbLightCtrl.bPIR
    Rectangle (77,54 122x22), "PIR status"
END_VISUALIZATION

// ---- POUs/Alle_Rum/Gange/Gang_4_210A/Visualization_4_307_1_1.TcVIS
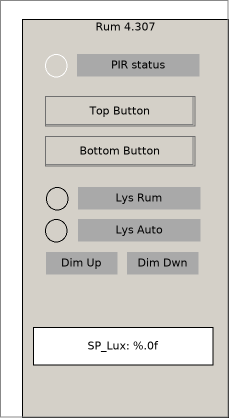
VISUALIZATION Visualization_4_307_1_1  // 229x418
    RoundedRectangle (22,19 207x399), "Rum 4.307"
    Rectangle (33,327 180x38), "SP_Lux: %.0f", text variable: P_Rum_4_307.fbLys.fbLightCtrl.fLuxZone1
    Button (45,96 150x30), "Top Button"
        tap P_Rum_4_307.bTopButtonZone1_Visu
    Button (45,136 150x30), "Bottom Button"
        tap P_Rum_4_307.bBottomButtonZone1_Visu
    Ellipse (46,187 22x23), colour toggle: P_Rum_4_307.fbLys.fbLightCtrl.bOnZone1
    Rectangle (78,187 122x22), "Lys Rum"
    Rectangle (46,252 71x22), "Dim Up", colour toggle: P_Rum_4_307.fbLys.fbLightCtrl.bDimUp
    Rectangle (127,252 71x22), "Dim Dwn", colour toggle: P_Rum_4_307.fbLys.fbLightCtrl.bDimDwn
    Ellipse (45,219 22x23), colour toggle: P_Rum_4_307.fbLys.fbLightCtrl.bAutoZone1
    Rectangle (78,219 122x22), "Lys Auto"
    Ellipse (45,54 22x23), colour toggle: P_Rum_4_307.fbLys.fbLightCtrl.bPIR
    Rectangle (77,54 122x22), "PIR status"
END_VISUALIZATION

// ---- POUs/Alle_Rum/Rum_Med_DALI_Pir/Rum_4_206/Visualization_5_338_1_1.TcVIS
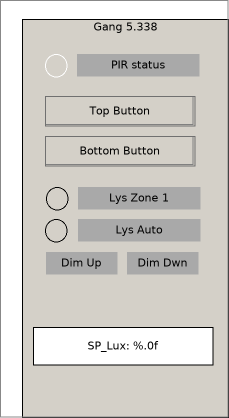
VISUALIZATION Visualization_5_338_1_1  // 229x418
    RoundedRectangle (22,19 207x399), "Gang 5.338"
    Rectangle (33,327 180x38), "SP_Lux: %.0f", text variable: P_Gang_5_338.arrfbLysGruppe[1].fbLightCtrl.fLuxZone1
    Button (45,96 150x30), "Top Button"
        tap P_Gang_5_338.bTopButtonZone1_Visu
    Button (45,136 150x30), "Bottom Button"
        tap P_Gang_5_338.bBottomButtonZone1_Visu
    Ellipse (46,187 22x23), colour toggle: P_Gang_5_338.arrfbLysGruppe[1].fbLightCtrl.bOnZone1
    Rectangle (78,187 122x22), "Lys Zone 1"
    Rectangle (46,252 71x22), "Dim Up", colour toggle: P_Gang_5_338.arrfbLysGruppe[1].fbLightCtrl.bDimUp
    Rectangle (127,252 71x22), "Dim Dwn", colour toggle: P_Gang_5_338.arrfbLysGruppe[1].fbLightCtrl.bDimDwn
    Ellipse (45,219 22x23), colour toggle: P_Gang_5_338.arrfbLysGruppe[1].fbLightCtrl.bAutoZone1
    Rectangle (78,219 122x22), "Lys Auto"
    Ellipse (45,54 22x23), colour toggle: P_Gang_5_338.arrfbLysGruppe[1].fbLightCtrl.bPIR
    Rectangle (77,54 122x22), "PIR status"
END_VISUALIZATION

// ---- POUs/Alle_Rum/Rum_Med_DALI_Pir/Rum_4_211A/Visualization_5_338_1_1_1.TcVIS
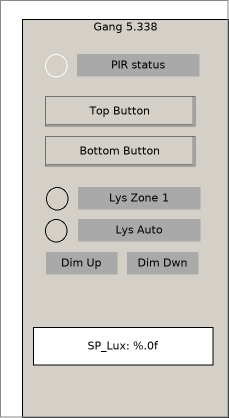
VISUALIZATION Visualization_5_338_1_1_1  // 229x418
    RoundedRectangle (22,19 207x399), "Gang 5.338"
    Rectangle (33,327 180x38), "SP_Lux: %.0f", text variable: P_Gang_5_338.arrfbLysGruppe[1].fbLightCtrl.fLuxZone1
    Button (45,96 150x30), "Top Button"
        tap P_Gang_5_338.bTopButtonZone1_Visu
    Button (45,136 150x30), "Bottom Button"
        tap P_Gang_5_338.bBottomButtonZone1_Visu
    Ellipse (46,187 22x23), colour toggle: P_Gang_5_338.arrfbLysGruppe[1].fbLightCtrl.bOnZone1
    Rectangle (78,187 122x22), "Lys Zone 1"
    Rectangle (46,252 71x22), "Dim Up", colour toggle: P_Gang_5_338.arrfbLysGruppe[1].fbLightCtrl.bDimUp
    Rectangle (127,252 71x22), "Dim Dwn", colour toggle: P_Gang_5_338.arrfbLysGruppe[1].fbLightCtrl.bDimDwn
    Ellipse (45,219 22x23), colour toggle: P_Gang_5_338.arrfbLysGruppe[1].fbLightCtrl.bAutoZone1
    Rectangle (78,219 122x22), "Lys Auto"
    Ellipse (45,54 22x23), colour toggle: P_Gang_5_338.arrfbLysGruppe[1].fbLightCtrl.bPIR
    Rectangle (77,54 122x22), "PIR status"
END_VISUALIZATION

// ---- POUs/Alle_Rum/Rum_Med_DALI_Pir/Rum_4_207/Visualization_4_307_1.TcVIS
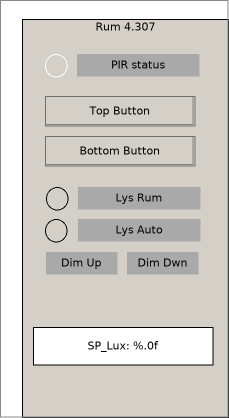
VISUALIZATION Visualization_4_307_1  // 229x418
    RoundedRectangle (22,19 207x399), "Rum 4.307"
    Rectangle (33,327 180x38), "SP_Lux: %.0f", text variable: P_Rum_4_307.fbLys.fbLightCtrl.fLuxZone1
    Button (45,96 150x30), "Top Button"
        tap P_Rum_4_307.bTopButtonZone1_Visu
    Button (45,136 150x30), "Bottom Button"
        tap P_Rum_4_307.bBottomButtonZone1_Visu
    Ellipse (46,187 22x23), colour toggle: P_Rum_4_307.fbLys.fbLightCtrl.bOnZone1
    Rectangle (78,187 122x22), "Lys Rum"
    Rectangle (46,252 71x22), "Dim Up", colour toggle: P_Rum_4_307.fbLys.fbLightCtrl.bDimUp
    Rectangle (127,252 71x22), "Dim Dwn", colour toggle: P_Rum_4_307.fbLys.fbLightCtrl.bDimDwn
    Ellipse (45,219 22x23), colour toggle: P_Rum_4_307.fbLys.fbLightCtrl.bAutoZone1
    Rectangle (78,219 122x22), "Lys Auto"
    Ellipse (45,54 22x23), colour toggle: P_Rum_4_307.fbLys.fbLightCtrl.bPIR
    Rectangle (77,54 122x22), "PIR status"
END_VISUALIZATION

// ---- POUs/DALI/DALI_Setup/VISUs/TextLists/CommandOnTerminalEvent.TcTLO
TEXTLIST CommandOnTerminalEvent
  0 = 'Do Nothing'
  1 = 'Off'
  2 = 'RecallMaxLevel'
  3 = 'RecallMinLevel'
  4 = 'GoToScene0'
  5 = 'GoToScene1'
  6 = 'GoToScene2'
  7 = 'GoToScene3'
  8 = 'GoToScene4'
  9 = 'GoToScene5'
  10 = 'GoToScene6'
  11 = 'GoToScene7'
  12 = 'GoToScene8'
  13 = 'GoToScene9'
  14 = 'GoToScene10'
  15 = 'GoToScene11'
  16 = 'GoToScene12'
  17 = 'GoToScene13'
  18 = 'GoToScene14'
  19 = 'GoToScene15'
   = ''
END_TEXTLIST

// ---- POUs/DALI/DALI_Setup/VISUs/TextLists/DimmingCurve.TcTLO
TEXTLIST DimmingCurve
  0 = 'Standard'
  1 = 'Linear'
  255 = 'Unknown'
   = ''
END_TEXTLIST

// ---- POUs/DALI/DALI_Setup/VISUs/TextLists/EventScheme.TcTLO
TEXTLIST EventScheme
  0 = '0 - Instance type and number'
  1 = '1 - Short address and instance type'
  2 = '2 - Short address and instance number'
  3 = '3 - Device group and instance type'
  4 = '4 - Instance group and instance type'
   = ''
END_TEXTLIST

// ---- POUs/DALI/DALI_Setup/VISUs/TextLists/FadeTime.TcTLO
TEXTLIST FadeTime
  0 = 'Extended Fade Time'
  1 = '0,7 s'
  2 = '1,0 s'
  3 = '1,4 s'
  4 = '2,0 s'
  5 = '2,8 s'
  6 = '4,0 s'
  7 = '5,7 s'
  8 = '8,0 s'
  9 = '11,3 s'
  10 = '16,0 s'
  11 = '22,6 s'
  12 = '32,0 s'
  13 = '45,3 s'
  14 = '64,0 s'
  15 = '90,5 s'
   = ''
END_TEXTLIST

// ---- POUs/DALI/DALI_Setup/VISUs/Visu_DALICommissioning.TcVIS
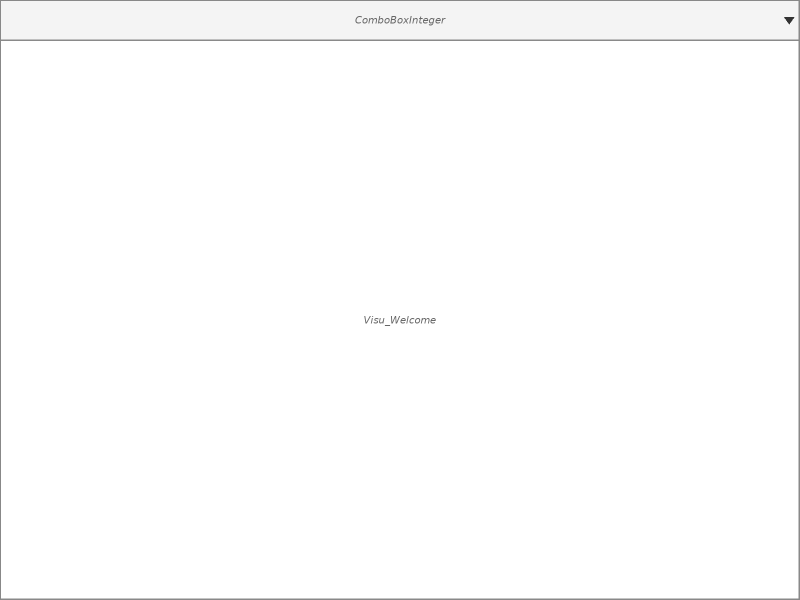
VISUALIZATION Visu_DALICommissioning  // 800x600
    ComboBoxInteger (0,0 800x40), variable: DALI_Commissioning.nSelectedDialog, input disabled if: DALI_Commissioning.bDisableComboBox, text list: 'TextList_Dialogs'
    Frame (0,40 800x560), frame switch variable: DALI_Commissioning.nSelectedDialog
        shows Visu_Welcome()
        shows Visu_Part102Commands()
        shows Visu_Part102Addressing()
        shows Visu_Part102Parameters()
        shows Visu_Part102Groups()
        shows Visu_Part102Scenes()
        shows Visu_Part102MemoryBank()
        shows Visu_Part102SetFading()
        shows Visu_Part202()
        shows Visu_Part205()
        shows Visu_Part207()
        shows Visu_Part208Switching()
        shows Visu_Part103Addressing()
        shows Visu_Part103Parameters()
        shows Visu_Part103Identify()
        shows Visu_Part301PushButton()
        shows Visu_Part302AbsoluteInputDevice()
        shows Visu_Part303OccupancySensor()
        shows Visu_Part304LightSensor()
        shows Visu_Part300GenericDevice()
        shows Visu_Part103MemoryBank()
        shows Visu_KL6821Configuration()
END_VISUALIZATION

// ---- POUs/DALI/DALI_Setup/VISUs/Visu_DALICommissioning/Visu_Part102Addressing.TcVIS
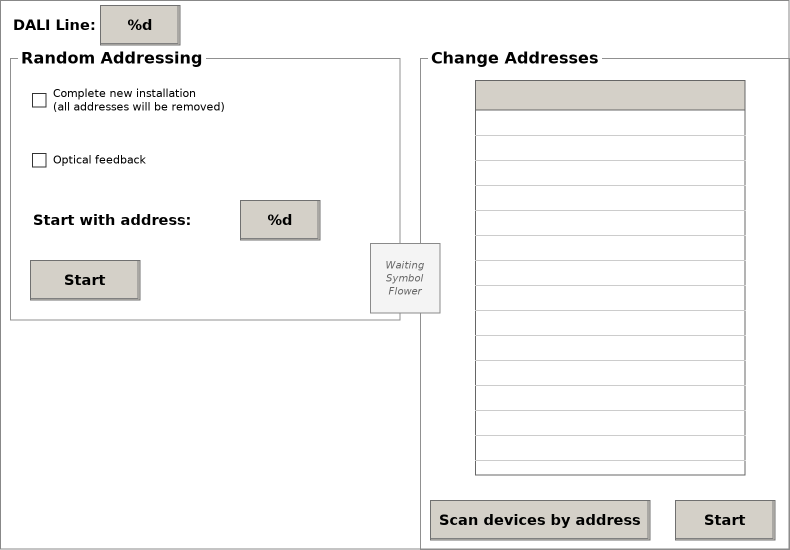
VISUALIZATION Visu_Part102Addressing  // 790x550
    GroupBox (420,50 370x500), "Change Addresses"
        Table (55,30 270x395), data array: DALI_Commissioning.fbPart102Addressing.aChangeAddressList
            p3854506369: DALI_Commissioning.fbPart102Addressing.aChangeAddressList[INDEX].nOldAddress
            p1892666644: DALI_Commissioning.fbPart102Addressing.aChangeAddressList[INDEX].nNewAddress
            p338671338: DALI_Commissioning.fbPart102Addressing.aChangeAddressList[INDEX].nRandomAddress
            p2170511999: DALI_Commissioning.fbPart102Addressing.aChangeAddressList[INDEX].nErrors
            Columns.Column.[0].Template: DALI_Commissioning.fbPart102Addressing.aNoShortAddress[INDEX]
            Columns.Column.[1].Template: DALI_Commissioning.fbPart102Addressing.aNoShortAddress[INDEX]; OnMouseClick: write the text variable via Default, min 0, max 63, title "New Short Address"
        Button (255,450 100x40), "Start"
            OnMouseClick: execute { DALI_Commissioning.fbPart102Addressing.bStartChangeAddress := TRUE; }
        Button (10,450 220x40), "Scan devices by address"
            OnMouseClick: execute { DALI_Commissioning.fbPart102Addressing.bScanDevices := TRUE; }
    GroupBox (10,50 390x270), "Random Addressing"
        Button (20,210 110x40), "Start"
            OnMouseClick: execute { DALI_Commissioning.fbPart102Addressing.bStartRandomAddressing := TRUE; }
        Checkbox (20,30 360x40), "Complete new installation (all addresses will be removed)", variable: DALI_Commissioning.fbPart102Addressing.bNewInstallation
        Checkbox (20,90 360x40), "Optical feedback", variable: DALI_Commissioning.fbPart102Addressing.bOpticalFeedback
        Textfield (20,150 200x40), "Start with address:"
        Button (230,150 80x40), "%d", text variable: DALI_Commissioning.fbPart102Addressing.nStartAddress
            OnMouseClick: write the text variable via Default, min 0, max 63, title "Insert Short Address"
    WaitingSymbolFlower (370,243 70x70), invisible if: DALI_Commissioning.fbPart102Addressing.bHideWaitSymbol
    Group (10,5 170x40)
        Textfield (0,0 110x40), "DALI Line:"
        Button (90,0 80x40), "%d", text variable: GVL_Internal.nDALILine
            OnMouseClick: write the text variable via Default, min 1, max 10, title "Choose line"
END_VISUALIZATION

// ---- POUs/DALI/DALI_Setup/VISUs/Visu_DALICommissioning/Visu_Part102Groups.TcVIS
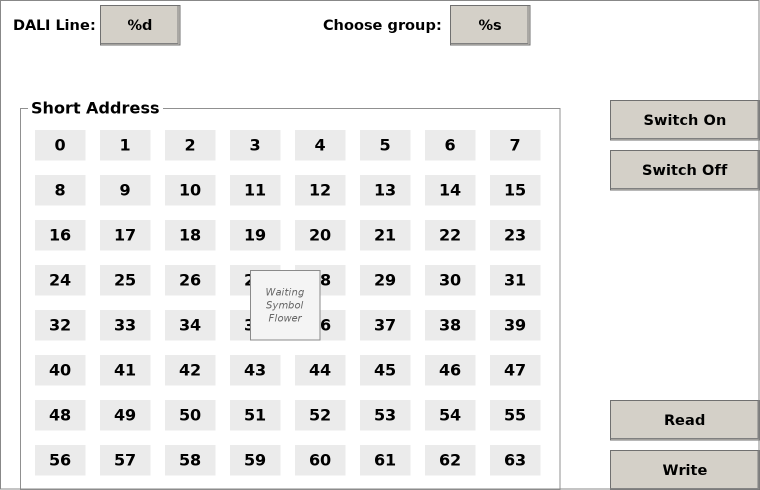
VISUALIZATION Visu_Part102Groups  // 760x490
    GroupBox (20,100 540x390), "Short Address"
        Textfield (15,30 50x30), "0", colour toggle: DALI_Commissioning.fbPart102Groups.aShowAlarmState[0] = TRUE, invisible if: DALI_Commissioning.fbPart102Groups.aActivateButton[0] = FALSE, input disabled if: DALI_Commissioning.fbPart102Groups.aActivateButton[0] = FALSE
            OnMouseClick: execute { DALI_Commissioning.fbPart102Groups.aButtonClick[0] := TRUE; }
        Textfield (80,30 50x30), "1", colour toggle: DALI_Commissioning.fbPart102Groups.aShowAlarmState[1] = TRUE, invisible if: DALI_Commissioning.fbPart102Groups.aActivateButton[1] = FALSE, input disabled if: DALI_Commissioning.fbPart102Groups.aActivateButton[1] = FALSE
            OnMouseClick: execute { DALI_Commissioning.fbPart102Groups.aButtonClick[1] := TRUE; }
        Textfield (145,30 50x30), "2", colour toggle: DALI_Commissioning.fbPart102Groups.aShowAlarmState[2] = TRUE, invisible if: DALI_Commissioning.fbPart102Groups.aActivateButton[2] = FALSE, input disabled if: DALI_Commissioning.fbPart102Groups.aActivateButton[2] = FALSE
            OnMouseClick: execute { DALI_Commissioning.fbPart102Groups.aButtonClick[2] := TRUE; }
        Textfield (210,30 50x30), "3", colour toggle: DALI_Commissioning.fbPart102Groups.aShowAlarmState[3] = TRUE, invisible if: DALI_Commissioning.fbPart102Groups.aActivateButton[3] = FALSE, input disabled if: DALI_Commissioning.fbPart102Groups.aActivateButton[3] = FALSE
            OnMouseClick: execute { DALI_Commissioning.fbPart102Groups.aButtonClick[3] := TRUE; }
        Textfield (275,30 50x30), "4", colour toggle: DALI_Commissioning.fbPart102Groups.aShowAlarmState[4] = TRUE, invisible if: DALI_Commissioning.fbPart102Groups.aActivateButton[4] = FALSE, input disabled if: DALI_Commissioning.fbPart102Groups.aActivateButton[4] = FALSE
            OnMouseClick: execute { DALI_Commissioning.fbPart102Groups.aButtonClick[4] := TRUE; }
        Textfield (340,30 50x30), "5", colour toggle: DALI_Commissioning.fbPart102Groups.aShowAlarmState[5] = TRUE, invisible if: DALI_Commissioning.fbPart102Groups.aActivateButton[5] = FALSE, input disabled if: DALI_Commissioning.fbPart102Groups.aActivateButton[5] = FALSE
            OnMouseClick: execute { DALI_Commissioning.fbPart102Groups.aButtonClick[5] := TRUE; }
        Textfield (405,30 50x30), "6", colour toggle: DALI_Commissioning.fbPart102Groups.aShowAlarmState[6] = TRUE, invisible if: DALI_Commissioning.fbPart102Groups.aActivateButton[6] = FALSE, input disabled if: DALI_Commissioning.fbPart102Groups.aActivateButton[6] = FALSE
            OnMouseClick: execute { DALI_Commissioning.fbPart102Groups.aButtonClick[6] := TRUE; }
        Textfield (470,30 50x30), "7", colour toggle: DALI_Commissioning.fbPart102Groups.aShowAlarmState[7] = TRUE, invisible if: DALI_Commissioning.fbPart102Groups.aActivateButton[7] = FALSE, input disabled if: DALI_Commissioning.fbPart102Groups.aActivateButton[7] = FALSE
            OnMouseClick: execute { DALI_Commissioning.fbPart102Groups.aButtonClick[7] := TRUE; }
        Textfield (15,75 50x30), "8", colour toggle: DALI_Commissioning.fbPart102Groups.aShowAlarmState[8] = TRUE, invisible if: DALI_Commissioning.fbPart102Groups.aActivateButton[8] = FALSE, input disabled if: DALI_Commissioning.fbPart102Groups.aActivateButton[8] = FALSE
            OnMouseClick: execute { DALI_Commissioning.fbPart102Groups.aButtonClick[8] := TRUE; }
        Textfield (80,75 50x30), "9", colour toggle: DALI_Commissioning.fbPart102Groups.aShowAlarmState[9] = TRUE, invisible if: DALI_Commissioning.fbPart102Groups.aActivateButton[9] = FALSE, input disabled if: DALI_Commissioning.fbPart102Groups.aActivateButton[9] = FALSE
            OnMouseClick: execute { DALI_Commissioning.fbPart102Groups.aButtonClick[9] := TRUE; }
        Textfield (145,75 50x30), "10", colour toggle: DALI_Commissioning.fbPart102Groups.aShowAlarmState[10] = TRUE, invisible if: DALI_Commissioning.fbPart102Groups.aActivateButton[10] = FALSE, input disabled if: DALI_Commissioning.fbPart102Groups.aActivateButton[10] = FALSE
            OnMouseClick: execute { DALI_Commissioning.fbPart102Groups.aButtonClick[10] := TRUE; }
        Textfield (210,75 50x30), "11", colour toggle: DALI_Commissioning.fbPart102Groups.aShowAlarmState[11] = TRUE, invisible if: DALI_Commissioning.fbPart102Groups.aActivateButton[11] = FALSE, input disabled if: DALI_Commissioning.fbPart102Groups.aActivateButton[11] = FALSE
            OnMouseClick: execute { DALI_Commissioning.fbPart102Groups.aButtonClick[11] := TRUE; }
        Textfield (275,75 50x30), "12", colour toggle: DALI_Commissioning.fbPart102Groups.aShowAlarmState[12] = TRUE, invisible if: DALI_Commissioning.fbPart102Groups.aActivateButton[12] = FALSE, input disabled if: DALI_Commissioning.fbPart102Groups.aActivateButton[12] = FALSE
            OnMouseClick: execute { DALI_Commissioning.fbPart102Groups.aButtonClick[12] := TRUE; }
        Textfield (340,75 50x30), "13", colour toggle: DALI_Commissioning.fbPart102Groups.aShowAlarmState[13] = TRUE, invisible if: DALI_Commissioning.fbPart102Groups.aActivateButton[13] = FALSE, input disabled if: DALI_Commissioning.fbPart102Groups.aActivateButton[13] = FALSE
            OnMouseClick: execute { DALI_Commissioning.fbPart102Groups.aButtonClick[13] := TRUE; }
        Textfield (405,75 50x30), "14", colour toggle: DALI_Commissioning.fbPart102Groups.aShowAlarmState[14] = TRUE, invisible if: DALI_Commissioning.fbPart102Groups.aActivateButton[14] = FALSE, input disabled if: DALI_Commissioning.fbPart102Groups.aActivateButton[14] = FALSE
            OnMouseClick: execute { DALI_Commissioning.fbPart102Groups.aButtonClick[14] := TRUE; }
        Textfield (470,75 50x30), "15", colour toggle: DALI_Commissioning.fbPart102Groups.aShowAlarmState[15] = TRUE, invisible if: DALI_Commissioning.fbPart102Groups.aActivateButton[15] = FALSE, input disabled if: DALI_Commissioning.fbPart102Groups.aActivateButton[15] = FALSE
            OnMouseClick: execute { DALI_Commissioning.fbPart102Groups.aButtonClick[15] := TRUE; }
        Textfield (15,120 50x30), "16", colour toggle: DALI_Commissioning.fbPart102Groups.aShowAlarmState[16] = TRUE, invisible if: DALI_Commissioning.fbPart102Groups.aActivateButton[16] = FALSE, input disabled if: DALI_Commissioning.fbPart102Groups.aActivateButton[16] = FALSE
            OnMouseClick: execute { DALI_Commissioning.fbPart102Groups.aButtonClick[16] := TRUE; }
        Textfield (80,120 50x30), "17", colour toggle: DALI_Commissioning.fbPart102Groups.aShowAlarmState[17] = TRUE, invisible if: DALI_Commissioning.fbPart102Groups.aActivateButton[17] = FALSE, input disabled if: DALI_Commissioning.fbPart102Groups.aActivateButton[17] = FALSE
            OnMouseClick: execute { DALI_Commissioning.fbPart102Groups.aButtonClick[17] := TRUE; }
        Textfield (145,120 50x30), "18", colour toggle: DALI_Commissioning.fbPart102Groups.aShowAlarmState[18] = TRUE, invisible if: DALI_Commissioning.fbPart102Groups.aActivateButton[18] = FALSE, input disabled if: DALI_Commissioning.fbPart102Groups.aActivateButton[18] = FALSE
            OnMouseClick: execute { DALI_Commissioning.fbPart102Groups.aButtonClick[18] := TRUE; }
        Textfield (210,120 50x30), "19", colour toggle: DALI_Commissioning.fbPart102Groups.aShowAlarmState[19] = TRUE, invisible if: DALI_Commissioning.fbPart102Groups.aActivateButton[19] = FALSE, input disabled if: DALI_Commissioning.fbPart102Groups.aActivateButton[19] = FALSE
            OnMouseClick: execute { DALI_Commissioning.fbPart102Groups.aButtonClick[19] := TRUE; }
        Textfield (275,120 50x30), "20", colour toggle: DALI_Commissioning.fbPart102Groups.aShowAlarmState[20] = TRUE, invisible if: DALI_Commissioning.fbPart102Groups.aActivateButton[20] = FALSE, input disabled if: DALI_Commissioning.fbPart102Groups.aActivateButton[20] = FALSE
            OnMouseClick: execute { DALI_Commissioning.fbPart102Groups.aButtonClick[20] := TRUE; }
        Textfield (340,120 50x30), "21", colour toggle: DALI_Commissioning.fbPart102Groups.aShowAlarmState[21] = TRUE, invisible if: DALI_Commissioning.fbPart102Groups.aActivateButton[21] = FALSE, input disabled if: DALI_Commissioning.fbPart102Groups.aActivateButton[21] = FALSE
            OnMouseClick: execute { DALI_Commissioning.fbPart102Groups.aButtonClick[21] := TRUE; }
        Textfield (405,120 50x30), "22", colour toggle: DALI_Commissioning.fbPart102Groups.aShowAlarmState[22] = TRUE, invisible if: DALI_Commissioning.fbPart102Groups.aActivateButton[22] = FALSE, input disabled if: DALI_Commissioning.fbPart102Groups.aActivateButton[22] = FALSE
            OnMouseClick: execute { DALI_Commissioning.fbPart102Groups.aButtonClick[22] := TRUE; }
        Textfield (470,120 50x30), "23", colour toggle: DALI_Commissioning.fbPart102Groups.aShowAlarmState[23] = TRUE, invisible if: DALI_Commissioning.fbPart102Groups.aActivateButton[23] = FALSE, input disabled if: DALI_Commissioning.fbPart102Groups.aActivateButton[23] = FALSE
            OnMouseClick: execute { DALI_Commissioning.fbPart102Groups.aButtonClick[23] := TRUE; }
        Textfield (15,165 50x30), "24", colour toggle: DALI_Commissioning.fbPart102Groups.aShowAlarmState[24] = TRUE, invisible if: DALI_Commissioning.fbPart102Groups.aDeviceGroupState[24] = 0, input disabled if: DALI_Commissioning.fbPart102Groups.aDeviceGroupState[24] = 0
            OnMouseClick: execute { DALI_Commissioning.fbPart102Groups.aButtonClick[24] := TRUE; }
        Textfield (80,165 50x30), "25", colour toggle: DALI_Commissioning.fbPart102Groups.aShowAlarmState[25] = TRUE, invisible if: DALI_Commissioning.fbPart102Groups.aActivateButton[25] = FALSE, input disabled if: DALI_Commissioning.fbPart102Groups.aActivateButton[25] = FALSE
            OnMouseClick: execute { DALI_Commissioning.fbPart102Groups.aButtonClick[25] := TRUE; }
        Textfield (145,165 50x30), "26", colour toggle: DALI_Commissioning.fbPart102Groups.aShowAlarmState[26] = TRUE, invisible if: DALI_Commissioning.fbPart102Groups.aActivateButton[26] = FALSE, input disabled if: DALI_Commissioning.fbPart102Groups.aActivateButton[26] = FALSE
            OnMouseClick: execute { DALI_Commissioning.fbPart102Groups.aButtonClick[26] := TRUE; }
        Textfield (210,165 50x30), "27", colour toggle: DALI_Commissioning.fbPart102Groups.aShowAlarmState[27] = TRUE, invisible if: DALI_Commissioning.fbPart102Groups.aActivateButton[27] = FALSE, input disabled if: DALI_Commissioning.fbPart102Groups.aActivateButton[27] = FALSE
            OnMouseClick: execute { DALI_Commissioning.fbPart102Groups.aButtonClick[27] := TRUE; }
        Textfield (275,165 50x30), "28", colour toggle: DALI_Commissioning.fbPart102Groups.aShowAlarmState[28] = TRUE, invisible if: DALI_Commissioning.fbPart102Groups.aActivateButton[28] = FALSE, input disabled if: DALI_Commissioning.fbPart102Groups.aActivateButton[28] = FALSE
            OnMouseClick: execute { DALI_Commissioning.fbPart102Groups.aButtonClick[28] := TRUE; }
        Textfield (340,165 50x30), "29", colour toggle: DALI_Commissioning.fbPart102Groups.aShowAlarmState[29] = TRUE, invisible if: DALI_Commissioning.fbPart102Groups.aActivateButton[29] = FALSE, input disabled if: DALI_Commissioning.fbPart102Groups.aActivateButton[29] = FALSE
            OnMouseClick: execute { DALI_Commissioning.fbPart102Groups.aButtonClick[29] := TRUE; }
        Textfield (405,165 50x30), "30", colour toggle: DALI_Commissioning.fbPart102Groups.aShowAlarmState[30] = TRUE, invisible if: DALI_Commissioning.fbPart102Groups.aActivateButton[30] = FALSE, input disabled if: DALI_Commissioning.fbPart102Groups.aActivateButton[30] = FALSE
            OnMouseClick: execute { DALI_Commissioning.fbPart102Groups.aButtonClick[30] := TRUE; }
        Textfield (470,165 50x30), "31", colour toggle: DALI_Commissioning.fbPart102Groups.aShowAlarmState[31] = TRUE, invisible if: DALI_Commissioning.fbPart102Groups.aActivateButton[31] = FALSE, input disabled if: DALI_Commissioning.fbPart102Groups.aActivateButton[31] = FALSE
            OnMouseClick: execute { DALI_Commissioning.fbPart102Groups.aButtonClick[31] := TRUE; }
        Textfield (15,210 50x30), "32", colour toggle: DALI_Commissioning.fbPart102Groups.aShowAlarmState[32] = TRUE, invisible if: DALI_Commissioning.fbPart102Groups.aActivateButton[32] = FALSE, input disabled if: DALI_Commissioning.fbPart102Groups.aActivateButton[32] = FALSE
            OnMouseClick: execute { DALI_Commissioning.fbPart102Groups.aButtonClick[32] := TRUE; }
        Textfield (80,210 50x30), "33", colour toggle: DALI_Commissioning.fbPart102Groups.aShowAlarmState[33] = TRUE, invisible if: DALI_Commissioning.fbPart102Groups.aActivateButton[33] = FALSE, input disabled if: DALI_Commissioning.fbPart102Groups.aActivateButton[33] = FALSE
            OnMouseClick: execute { DALI_Commissioning.fbPart102Groups.aButtonClick[33] := TRUE; }
        Textfield (145,210 50x30), "34", colour toggle: DALI_Commissioning.fbPart102Groups.aShowAlarmState[34] = TRUE, invisible if: DALI_Commissioning.fbPart102Groups.aActivateButton[34] = FALSE, input disabled if: DALI_Commissioning.fbPart102Groups.aActivateButton[34] = FALSE
            OnMouseClick: execute { DALI_Commissioning.fbPart102Groups.aButtonClick[34] := TRUE; }
        Textfield (210,210 50x30), "35", colour toggle: DALI_Commissioning.fbPart102Groups.aShowAlarmState[35] = TRUE, invisible if: DALI_Commissioning.fbPart102Groups.aActivateButton[35] = FALSE, input disabled if: DALI_Commissioning.fbPart102Groups.aActivateButton[35] = FALSE
            OnMouseClick: execute { DALI_Commissioning.fbPart102Groups.aButtonClick[35] := TRUE; }
        Textfield (275,210 50x30), "36", colour toggle: DALI_Commissioning.fbPart102Groups.aShowAlarmState[36] = TRUE, invisible if: DALI_Commissioning.fbPart102Groups.aActivateButton[36] = FALSE, input disabled if: DALI_Commissioning.fbPart102Groups.aActivateButton[36] = FALSE
            OnMouseClick: execute { DALI_Commissioning.fbPart102Groups.aButtonClick[36] := TRUE; }
        Textfield (340,210 50x30), "37", colour toggle: DALI_Commissioning.fbPart102Groups.aShowAlarmState[37] = TRUE, invisible if: DALI_Commissioning.fbPart102Groups.aActivateButton[37] = FALSE, input disabled if: DALI_Commissioning.fbPart102Groups.aActivateButton[37] = FALSE
            OnMouseClick: execute { DALI_Commissioning.fbPart102Groups.aButtonClick[37] := TRUE; }
        Textfield (405,210 50x30), "38", colour toggle: DALI_Commissioning.fbPart102Groups.aShowAlarmState[38] = TRUE, invisible if: DALI_Commissioning.fbPart102Groups.aActivateButton[38] = FALSE, input disabled if: DALI_Commissioning.fbPart102Groups.aActivateButton[38] = FALSE
            OnMouseClick: execute { DALI_Commissioning.fbPart102Groups.aButtonClick[38] := TRUE; }
        Textfield (470,210 50x30), "39", colour toggle: DALI_Commissioning.fbPart102Groups.aShowAlarmState[39] = TRUE, invisible if: DALI_Commissioning.fbPart102Groups.aActivateButton[39] = FALSE, input disabled if: DALI_Commissioning.fbPart102Groups.aActivateButton[39] = FALSE
            OnMouseClick: execute { DALI_Commissioning.fbPart102Groups.aButtonClick[39] := TRUE; }
        Textfield (15,255 50x30), "40", colour toggle: DALI_Commissioning.fbPart102Groups.aShowAlarmState[40] = TRUE, invisible if: DALI_Commissioning.fbPart102Groups.aActivateButton[40] = FALSE, input disabled if: DALI_Commissioning.fbPart102Groups.aActivateButton[40] = FALSE
            OnMouseClick: execute { DALI_Commissioning.fbPart102Groups.aButtonClick[40] := TRUE; }
        Textfield (80,255 50x30), "41", colour toggle: DALI_Commissioning.fbPart102Groups.aShowAlarmState[41] = TRUE, invisible if: DALI_Commissioning.fbPart102Groups.aActivateButton[41] = FALSE, input disabled if: DALI_Commissioning.fbPart102Groups.aActivateButton[41] = FALSE
            OnMouseClick: execute { DALI_Commissioning.fbPart102Groups.aButtonClick[41] := TRUE; }
        Textfield (145,255 50x30), "42", colour toggle: DALI_Commissioning.fbPart102Groups.aShowAlarmState[42] = TRUE, invisible if: DALI_Commissioning.fbPart102Groups.aActivateButton[42] = FALSE, input disabled if: DALI_Commissioning.fbPart102Groups.aActivateButton[42] = FALSE
            OnMouseClick: execute { DALI_Commissioning.fbPart102Groups.aButtonClick[42] := TRUE; }
        Textfield (210,255 50x30), "43", colour toggle: DALI_Commissioning.fbPart102Groups.aShowAlarmState[43] = TRUE, invisible if: DALI_Commissioning.fbPart102Groups.aActivateButton[43] = FALSE, input disabled if: DALI_Commissioning.fbPart102Groups.aActivateButton[43] = FALSE
            OnMouseClick: execute { DALI_Commissioning.fbPart102Groups.aButtonClick[43] := TRUE; }
        Textfield (275,255 50x30), "44", colour toggle: DALI_Commissioning.fbPart102Groups.aShowAlarmState[44] = TRUE, invisible if: DALI_Commissioning.fbPart102Groups.aActivateButton[44] = FALSE, input disabled if: DALI_Commissioning.fbPart102Groups.aActivateButton[44] = FALSE
            OnMouseClick: execute { DALI_Commissioning.fbPart102Groups.aButtonClick[44] := TRUE; }
        Textfield (340,255 50x30), "45", colour toggle: DALI_Commissioning.fbPart102Groups.aShowAlarmState[45] = TRUE, invisible if: DALI_Commissioning.fbPart102Groups.aActivateButton[45] = FALSE, input disabled if: DALI_Commissioning.fbPart102Groups.aActivateButton[45] = FALSE
            OnMouseClick: execute { DALI_Commissioning.fbPart102Groups.aButtonClick[45] := TRUE; }
        Textfield (405,255 50x30), "46", colour toggle: DALI_Commissioning.fbPart102Groups.aShowAlarmState[46] = TRUE, invisible if: DALI_Commissioning.fbPart102Groups.aActivateButton[46] = FALSE, input disabled if: DALI_Commissioning.fbPart102Groups.aActivateButton[46] = FALSE
            OnMouseClick: execute { DALI_Commissioning.fbPart102Groups.aButtonClick[46] := TRUE; }
        Textfield (470,255 50x30), "47", colour toggle: DALI_Commissioning.fbPart102Groups.aShowAlarmState[47] = TRUE, invisible if: DALI_Commissioning.fbPart102Groups.aActivateButton[47] = FALSE, input disabled if: DALI_Commissioning.fbPart102Groups.aActivateButton[47] = FALSE
            OnMouseClick: execute { DALI_Commissioning.fbPart102Groups.aButtonClick[47] := TRUE; }
        Textfield (15,300 50x30), "48", colour toggle: DALI_Commissioning.fbPart102Groups.aShowAlarmState[48] = TRUE, invisible if: DALI_Commissioning.fbPart102Groups.aActivateButton[48] = FALSE, input disabled if: DALI_Commissioning.fbPart102Groups.aActivateButton[48] = FALSE
            OnMouseClick: execute { DALI_Commissioning.fbPart102Groups.aButtonClick[48] := TRUE; }
        Textfield (80,300 50x30), "49", colour toggle: DALI_Commissioning.fbPart102Groups.aShowAlarmState[49] = TRUE, invisible if: DALI_Commissioning.fbPart102Groups.aActivateButton[49] = FALSE, input disabled if: DALI_Commissioning.fbPart102Groups.aActivateButton[49] = FALSE
            OnMouseClick: execute { DALI_Commissioning.fbPart102Groups.aButtonClick[49] := TRUE; }
        Textfield (145,300 50x30), "50", colour toggle: DALI_Commissioning.fbPart102Groups.aShowAlarmState[50] = TRUE, invisible if: DALI_Commissioning.fbPart102Groups.aActivateButton[50] = FALSE, input disabled if: DALI_Commissioning.fbPart102Groups.aActivateButton[50] = FALSE
            OnMouseClick: execute { DALI_Commissioning.fbPart102Groups.aButtonClick[50] := TRUE; }
        Textfield (210,300 50x30), "51", colour toggle: DALI_Commissioning.fbPart102Groups.aShowAlarmState[51] = TRUE, invisible if: DALI_Commissioning.fbPart102Groups.aActivateButton[51] = FALSE, input disabled if: DALI_Commissioning.fbPart102Groups.aActivateButton[51] = FALSE
            OnMouseClick: execute { DALI_Commissioning.fbPart102Groups.aButtonClick[51] := TRUE; }
        Textfield (275,300 50x30), "52", colour toggle: DALI_Commissioning.fbPart102Groups.aShowAlarmState[52] = TRUE, invisible if: DALI_Commissioning.fbPart102Groups.aActivateButton[52] = FALSE, input disabled if: DALI_Commissioning.fbPart102Groups.aActivateButton[52] = FALSE
            OnMouseClick: execute { DALI_Commissioning.fbPart102Groups.aButtonClick[52] := TRUE; }
        Textfield (340,300 50x30), "53", colour toggle: DALI_Commissioning.fbPart102Groups.aShowAlarmState[53] = TRUE, invisible if: DALI_Commissioning.fbPart102Groups.aActivateButton[53] = FALSE, input disabled if: DALI_Commissioning.fbPart102Groups.aActivateButton[53] = FALSE
            OnMouseClick: execute { DALI_Commissioning.fbPart102Groups.aButtonClick[53] := TRUE; }
        Textfield (405,300 50x30), "54", colour toggle: DALI_Commissioning.fbPart102Groups.aShowAlarmState[54] = TRUE, invisible if: DALI_Commissioning.fbPart102Groups.aActivateButton[54] = FALSE, input disabled if: DALI_Commissioning.fbPart102Groups.aActivateButton[54] = FALSE
            OnMouseClick: execute { DALI_Commissioning.fbPart102Groups.aButtonClick[54] := TRUE; }
        Textfield (470,300 50x30), "55", colour toggle: DALI_Commissioning.fbPart102Groups.aShowAlarmState[55] = TRUE, invisible if: DALI_Commissioning.fbPart102Groups.aActivateButton[55] = FALSE, input disabled if: DALI_Commissioning.fbPart102Groups.aActivateButton[55] = FALSE
            OnMouseClick: execute { DALI_Commissioning.fbPart102Groups.aButtonClick[55] := TRUE; }
        Textfield (15,345 50x30), "56", colour toggle: DALI_Commissioning.fbPart102Groups.aShowAlarmState[56] = TRUE, invisible if: DALI_Commissioning.fbPart102Groups.aActivateButton[56] = FALSE, input disabled if: DALI_Commissioning.fbPart102Groups.aActivateButton[56] = FALSE
            OnMouseClick: execute { DALI_Commissioning.fbPart102Groups.aButtonClick[56] := TRUE; }
        Textfield (80,345 50x30), "57", colour toggle: DALI_Commissioning.fbPart102Groups.aShowAlarmState[57] = TRUE, invisible if: DALI_Commissioning.fbPart102Groups.aActivateButton[57] = FALSE, input disabled if: DALI_Commissioning.fbPart102Groups.aActivateButton[57] = FALSE
            OnMouseClick: execute { DALI_Commissioning.fbPart102Groups.aButtonClick[56] := TRUE; }
        Textfield (145,345 50x30), "58", colour toggle: DALI_Commissioning.fbPart102Groups.aShowAlarmState[58] = TRUE, invisible if: DALI_Commissioning.fbPart102Groups.aActivateButton[58] = FALSE, input disabled if: DALI_Commissioning.fbPart102Groups.aActivateButton[58] = FALSE
            OnMouseClick: execute { DALI_Commissioning.fbPart102Groups.aButtonClick[58] := TRUE; }
        Textfield (210,345 50x30), "59", colour toggle: DALI_Commissioning.fbPart102Groups.aShowAlarmState[59] = TRUE, invisible if: DALI_Commissioning.fbPart102Groups.aActivateButton[59] = FALSE, input disabled if: DALI_Commissioning.fbPart102Groups.aActivateButton[59] = FALSE
            OnMouseClick: execute { DALI_Commissioning.fbPart102Groups.aButtonClick[59] := TRUE; }
        Textfield (275,345 50x30), "60", colour toggle: DALI_Commissioning.fbPart102Groups.aShowAlarmState[60] = TRUE, invisible if: DALI_Commissioning.fbPart102Groups.aActivateButton[60] = FALSE, input disabled if: DALI_Commissioning.fbPart102Groups.aActivateButton[60] = FALSE
            OnMouseClick: execute { DALI_Commissioning.fbPart102Groups.aButtonClick[60] := TRUE; }
        Textfield (340,345 50x30), "61", colour toggle: DALI_Commissioning.fbPart102Groups.aShowAlarmState[61] = TRUE, invisible if: DALI_Commissioning.fbPart102Groups.aActivateButton[61] = FALSE, input disabled if: DALI_Commissioning.fbPart102Groups.aActivateButton[61] = FALSE
            OnMouseClick: execute { DALI_Commissioning.fbPart102Groups.aButtonClick[61] := TRUE; }
        Textfield (405,345 50x30), "62", colour toggle: DALI_Commissioning.fbPart102Groups.aShowAlarmState[62] = TRUE, invisible if: DALI_Commissioning.fbPart102Groups.aActivateButton[62] = FALSE, input disabled if: DALI_Commissioning.fbPart102Groups.aActivateButton[62] = FALSE
            OnMouseClick: execute { DALI_Commissioning.fbPart102Groups.aButtonClick[62] := TRUE; }
        Textfield (470,345 50x30), "63", colour toggle: DALI_Commissioning.fbPart102Groups.aShowAlarmState[63] = TRUE, invisible if: DALI_Commissioning.fbPart102Groups.aActivateButton[63] = FALSE, input disabled if: DALI_Commissioning.fbPart102Groups.aActivateButton[63] = FALSE
            OnMouseClick: execute { DALI_Commissioning.fbPart102Groups.aButtonClick[63] := TRUE; }
        WaitingSymbolFlower (230,170 70x70), invisible if: DALI_Commissioning.fbPart102Groups.bHideWaitSymbol
    Button (610,400 150x40), "Read"
        OnMouseClick: execute { DALI_Commissioning.fbPart102Groups.bRead := TRUE; }
    Button (610,450 150x40), "Write"
        OnMouseClick: execute { DALI_Commissioning.fbPart102Groups.bWrite := TRUE; }
    Button (610,100 150x40), "Switch On"
        OnMouseClick: execute { DALI_Commissioning.fbPart102Groups.bSwitchOn := TRUE; }
    Button (610,150 150x40), "Switch Off"
        OnMouseClick: execute { DALI_Commissioning.fbPart102Groups.bSwitchOff := TRUE; }
    Group (320,5 210x40)
        Textfield (0,0 120x40), "Choose group:"
        Button (130,0 80x40), "%s", text variable: DALI_Commissioning.fbPart102Groups.nGroupAddress
            OnMouseClick: write the text variable via Default, min 0, max 15, title "Choose group"
    Group (10,5 170x40)
        Textfield (0,0 110x40), "DALI Line:"
        Button (90,0 80x40), "%d", text variable: GVL_Internal.nDALILine
            OnMouseClick: write the text variable via Default, min 1, max 10, title "Choose line"
END_VISUALIZATION

// ---- POUs/DALI/DALI_Setup/VISUs/Visu_DALICommissioning/Visu_Part102Parameters.TcVIS
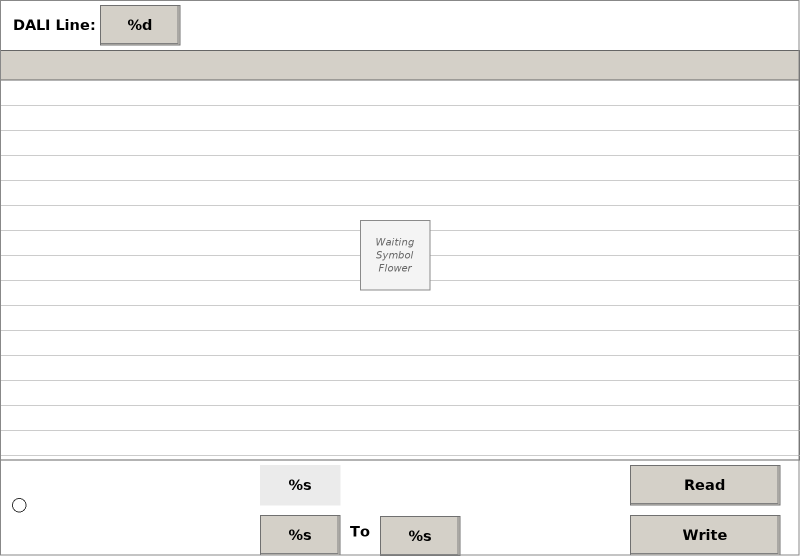
VISUALIZATION Visu_Part102Parameters  // 800x556
    Table (0,50 800x410), data array: DALI_Commissioning.fbPart102Parameters.aParameters
        p1137915858: DALI_Commissioning.fbPart102Parameters.nSelectedAddress
        p3854506369: DALI_Commissioning.fbPart102Parameters.aParameters[INDEX].nShortAddress
        p1892666644: DALI_Commissioning.fbPart102Parameters.aParameters[INDEX].nActualLevel
        p338671338: DALI_Commissioning.fbPart102Parameters.aParameters[INDEX].nMinLevel
        p2170511999: DALI_Commissioning.fbPart102Parameters.aParameters[INDEX].nMaxLevel
        p3723444502: DALI_Commissioning.fbPart102Parameters.aParameters[INDEX].eFadeRate
        p1218418051: DALI_Commissioning.fbPart102Parameters.aParameters[INDEX].eFadeTime
        p746581629: DALI_Commissioning.fbPart102Parameters.aParameters[INDEX].nPowerOnLevel
        p3104783080: DALI_Commissioning.fbPart102Parameters.aParameters[INDEX].nSystemFailureLevel
        p2501879983: DALI_Commissioning.fbPart102Parameters.aParameters[INDEX].nPhysicalMinimum
        p7306298: DALI_Commissioning.fbPart102Parameters.aParameters[INDEX].sDeviceTypes
        Columns.Column.[1].Template: OnMouseClick: write the text variable via Default, min 0, max 254, title "MinLevel"
        Columns.Column.[2].Template: OnMouseClick: write the text variable via Default, min 1, max 254, title "MaxLevel"
        Columns.Column.[3].Template: OnMouseClick: write the text variable via Default, min 0, max 254, title "FadeRate"
        Columns.Column.[4].Template: OnMouseClick: write the text variable via Default, min 1, max 15, title "Fade Rate"
        Columns.Column.[5].Template: OnMouseClick: write the text variable via Default, min 0, max 15, title "Fade Time"
        Columns.Column.[6].Template: OnMouseClick: write the text variable via Default, min 1, max 254, title "Power On Level"
        Columns.Column.[7].Template: OnMouseClick: write the text variable via Default, min 0, max 255, title "System Failure Level"
    RadioButton (10,455 254x100), variable: DALI_Commissioning.fbPart102Parameters.nAddressRange
        Areas[0]: Text=Single Short Address
        Areas[1]: Text=Short Address Range
    Textfield (335,516 50x31), "To"
    Button (630,465 150x40), "Read"
        OnMouseClick: execute { DALI_Commissioning.fbPart102Parameters.bRead := TRUE; }
    Button (630,515 150x40), "Write"
        OnMouseClick: execute { DALI_Commissioning.fbPart102Parameters.bWrite := TRUE; }
    Button (260,515 80x40), "%s", text variable: DALI_Commissioning.fbPart102Parameters.nStartAddress
        OnMouseClick: write the text variable via Default, min 0, max 63, title "Insert Short Address"
    Button (380,516 80x40), "%s", text variable: DALI_Commissioning.fbPart102Parameters.nEndAddress
        OnMouseClick: write the text variable via Default, min 0, max 63, title "Insert Short Address"
    Textfield (260,465 80x40), "%s", tooltip "Please select the desired Short Address in the table above.", text variable: DALI_Commissioning.fbPart102Parameters.nSelectedAddress
    WaitingSymbolFlower (360,220 70x70), invisible if: DALI_Commissioning.fbPart102Parameters.bHideWaitSymbol
    Group (10,5 170x40)
        Textfield (0,0 110x40), "DALI Line:"
        Button (90,0 80x40), "%d", text variable: GVL_Internal.nDALILine
            OnMouseClick: write the text variable via Default, min 1, max 10, title "Choose line"
END_VISUALIZATION

// ---- POUs/DALI/DALI_Setup/VISUs/Visu_DALICommissioning/Visu_Part102Scenes.TcVIS
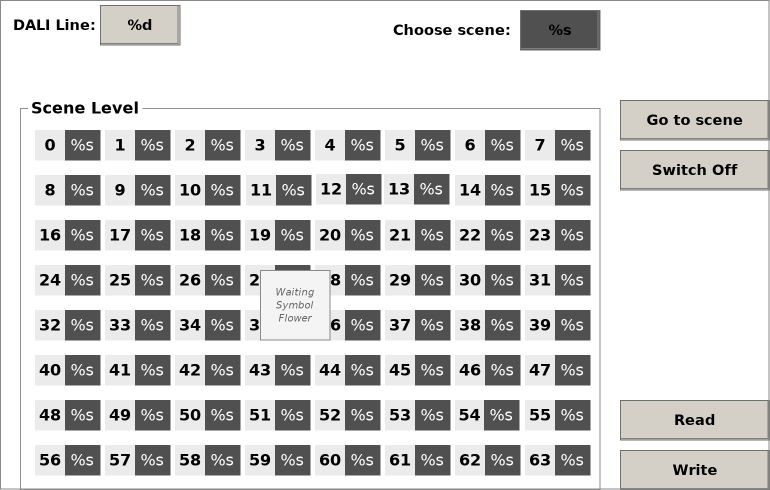
VISUALIZATION Visu_Part102Scenes  // 770x490
    GroupBox (20,100 580x390), "Scene Level"
        Group (85,30 65x30)
            Textfield (0,0 30x30), "1"
            Textfield (30,0 35x30), "%s", text variable: DALI_Commissioning.fbPart102Scenes.aScene[1], input disabled if: DALI_Commissioning.fbPart102Scenes.aNoShortAddress[1]
                p55702900: DALI_Commissioning.fbPart102Scenes.aFont[1]
                OnMouseClick: write the text variable via Default, min 0, max 255, title "Scene Value"
        Group (505,30 65x30)
            Textfield (0,0 30x30), "7"
            Textfield (30,0 35x30), "%s", text variable: DALI_Commissioning.fbPart102Scenes.aScene[7], input disabled if: DALI_Commissioning.fbPart102Scenes.aNoShortAddress[7]
                p55702900: DALI_Commissioning.fbPart102Scenes.aFont[7]
                OnMouseClick: write the text variable via Default, min 0, max 255, title "Scene Value"
        Group (435,30 65x30)
            Textfield (0,0 30x30), "6"
            Textfield (30,0 35x30), "%s", text variable: DALI_Commissioning.fbPart102Scenes.aScene[6], input disabled if: DALI_Commissioning.fbPart102Scenes.aNoShortAddress[6]
                p55702900: DALI_Commissioning.fbPart102Scenes.aFont[6]
                OnMouseClick: write the text variable via Default, min 0, max 255, title "Scene Value"
        Group (365,30 65x30)
            Textfield (0,0 30x30), "5"
            Textfield (30,0 35x30), "%s", text variable: DALI_Commissioning.fbPart102Scenes.aScene[5], input disabled if: DALI_Commissioning.fbPart102Scenes.aNoShortAddress[5]
                p55702900: DALI_Commissioning.fbPart102Scenes.aFont[5]
                OnMouseClick: write the text variable via Default, min 0, max 255, title "Scene Value"
        Group (295,30 65x30)
            Textfield (0,0 30x30), "4"
            Textfield (30,0 35x30), "%s", text variable: DALI_Commissioning.fbPart102Scenes.aScene[4], input disabled if: DALI_Commissioning.fbPart102Scenes.aNoShortAddress[4]
                p55702900: DALI_Commissioning.fbPart102Scenes.aFont[4]
                OnMouseClick: write the text variable via Default, min 0, max 255, title "Scene Value"
        Group (225,30 65x30)
            Textfield (0,0 30x30), "3"
            Textfield (30,0 35x30), "%s", text variable: DALI_Commissioning.fbPart102Scenes.aScene[3], input disabled if: DALI_Commissioning.fbPart102Scenes.aNoShortAddress[3]
                p55702900: DALI_Commissioning.fbPart102Scenes.aFont[3]
                OnMouseClick: write the text variable via Default, min 0, max 255, title "Scene Value"
        Group (155,30 65x30)
            Textfield (0,0 30x30), "2"
            Textfield (30,0 35x30), "%s", text variable: DALI_Commissioning.fbPart102Scenes.aScene[2], input disabled if: DALI_Commissioning.fbPart102Scenes.aNoShortAddress[2]
                p55702900: DALI_Commissioning.fbPart102Scenes.aFont[2]
                OnMouseClick: write the text variable via Default, min 0, max 255, title "Scene Value"
        Group (15,75 65x30)
            Textfield (0,0 30x30), "8"
            Textfield (30,0 35x30), "%s", text variable: DALI_Commissioning.fbPart102Scenes.aScene[8], input disabled if: DALI_Commissioning.fbPart102Scenes.aNoShortAddress[8]
                p55702900: DALI_Commissioning.fbPart102Scenes.aFont[8]
                OnMouseClick: write the text variable via Default, min 0, max 255, title "Scene Value"
        Group (15,120 65x30)
            Textfield (0,0 30x30), "16"
            Textfield (30,0 35x30), "%s", text variable: DALI_Commissioning.fbPart102Scenes.aScene[16], input disabled if: DALI_Commissioning.fbPart102Scenes.aNoShortAddress[16]
                p55702900: DALI_Commissioning.fbPart102Scenes.aFont[16]
                OnMouseClick: write the text variable via Default, min 0, max 255, title "Scene Value"
        Group (15,165 65x30)
            Textfield (0,0 30x30), "24"
            Textfield (30,0 35x30), "%s", text variable: DALI_Commissioning.fbPart102Scenes.aScene[24], input disabled if: DALI_Commissioning.fbPart102Scenes.aNoShortAddress[24]
                p55702900: DALI_Commissioning.fbPart102Scenes.aFont[24]
                OnMouseClick: write the text variable via Default, min 0, max 255, title "Scene Value"
        Group (15,210 65x30)
            Textfield (0,0 30x30), "32"
            Textfield (30,0 35x30), "%s", text variable: DALI_Commissioning.fbPart102Scenes.aScene[32], input disabled if: DALI_Commissioning.fbPart102Scenes.aNoShortAddress[32]
                p55702900: DALI_Commissioning.fbPart102Scenes.aFont[32]
                OnMouseClick: write the text variable via Default, min 0, max 255, title "Scene Value"
        Group (15,255 65x30)
            Textfield (0,0 30x30), "40"
            Textfield (30,0 35x30), "%s", text variable: DALI_Commissioning.fbPart102Scenes.aScene[40], input disabled if: DALI_Commissioning.fbPart102Scenes.aNoShortAddress[40]
                p55702900: DALI_Commissioning.fbPart102Scenes.aFont[40]
                OnMouseClick: write the text variable via Default, min 0, max 255, title "Scene Value"
        Group (15,300 65x30)
            Textfield (0,0 30x30), "48"
            Textfield (30,0 35x30), "%s", text variable: DALI_Commissioning.fbPart102Scenes.aScene[48], input disabled if: DALI_Commissioning.fbPart102Scenes.aNoShortAddress[48]
                p55702900: DALI_Commissioning.fbPart102Scenes.aFont[48]
                OnMouseClick: write the text variable via Default, min 0, max 255, title "Scene Value"
        Group (15,345 65x30)
            Textfield (0,0 30x30), "56"
            Textfield (30,0 35x30), "%s", text variable: DALI_Commissioning.fbPart102Scenes.aScene[56], input disabled if: DALI_Commissioning.fbPart102Scenes.aNoShortAddress[56]
                p55702900: DALI_Commissioning.fbPart102Scenes.aFont[56]
                OnMouseClick: write the text variable via Default, min 0, max 255, title "Scene Value"
        Group (85,75 65x30)
            Textfield (0,0 30x30), "9"
            Textfield (30,0 35x30), "%s", text variable: DALI_Commissioning.fbPart102Scenes.aScene[9], input disabled if: DALI_Commissioning.fbPart102Scenes.aNoShortAddress[9]
                p55702900: DALI_Commissioning.fbPart102Scenes.aFont[9]
                OnMouseClick: write the text variable via Default, min 0, max 255, title "Scene Value"
        Group (155,75 65x30)
            Textfield (0,0 30x30), "10"
            Textfield (30,0 35x30), "%s", text variable: DALI_Commissioning.fbPart102Scenes.aScene[10], input disabled if: DALI_Commissioning.fbPart102Scenes.aNoShortAddress[10]
                p55702900: DALI_Commissioning.fbPart102Scenes.aFont[10]
                OnMouseClick: write the text variable via Default, min 0, max 255, title "Scene Value"
        Group (226,75 65x30)
            Textfield (0,0 30x30), "11"
            Textfield (30,0 35x30), "%s", text variable: DALI_Commissioning.fbPart102Scenes.aScene[11], input disabled if: DALI_Commissioning.fbPart102Scenes.aNoShortAddress[11]
                p55702900: DALI_Commissioning.fbPart102Scenes.aFont[11]
                OnMouseClick: write the text variable via Default, min 0, max 255, title "Scene Value"
        Group (296,74 65x30)
            Textfield (0,0 30x30), "12"
            Textfield (30,0 35x30), "%s", text variable: DALI_Commissioning.fbPart102Scenes.aScene[12], input disabled if: DALI_Commissioning.fbPart102Scenes.aNoShortAddress[12]
                p55702900: DALI_Commissioning.fbPart102Scenes.aFont[12]
                OnMouseClick: write the text variable via Default, min 0, max 255, title "Scene Value"
        Group (364,74 65x30)
            Textfield (0,0 30x30), "13"
            Textfield (30,0 35x30), "%s", text variable: DALI_Commissioning.fbPart102Scenes.aScene[13], input disabled if: DALI_Commissioning.fbPart102Scenes.aNoShortAddress[13]
                p55702900: DALI_Commissioning.fbPart102Scenes.aFont[13]
                OnMouseClick: write the text variable via Default, min 0, max 255, title "Scene Value"
        Group (435,75 65x30)
            Textfield (0,0 30x30), "14"
            Textfield (30,0 35x30), "%s", text variable: DALI_Commissioning.fbPart102Scenes.aScene[14], input disabled if: DALI_Commissioning.fbPart102Scenes.aNoShortAddress[14]
                p55702900: DALI_Commissioning.fbPart102Scenes.aFont[14]
                OnMouseClick: write the text variable via Default, min 0, max 255, title "Scene Value"
        Group (505,75 65x30)
            Textfield (0,0 30x30), "15"
            Textfield (30,0 35x30), "%s", text variable: DALI_Commissioning.fbPart102Scenes.aScene[15], input disabled if: DALI_Commissioning.fbPart102Scenes.aNoShortAddress[15]
                p55702900: DALI_Commissioning.fbPart102Scenes.aFont[15]
                OnMouseClick: write the text variable via Default, min 0, max 255, title "Scene Value"
        Group (85,120 65x30)
            Textfield (0,0 30x30), "17"
            Textfield (30,0 35x30), "%s", text variable: DALI_Commissioning.fbPart102Scenes.aScene[17], input disabled if: DALI_Commissioning.fbPart102Scenes.aNoShortAddress[17]
                p55702900: DALI_Commissioning.fbPart102Scenes.aFont[17]
                OnMouseClick: write the text variable via Default, min 0, max 255, title "Scene Value"
        Group (155,120 65x30)
            Textfield (0,0 30x30), "18"
            Textfield (30,0 35x30), "%s", text variable: DALI_Commissioning.fbPart102Scenes.aScene[18], input disabled if: DALI_Commissioning.fbPart102Scenes.aNoShortAddress[18]
                p55702900: DALI_Commissioning.fbPart102Scenes.aFont[18]
                OnMouseClick: write the text variable via Default, min 0, max 255, title "Scene Value"
        Group (225,120 65x30)
            Textfield (0,0 30x30), "19"
            Textfield (30,0 35x30), "%s", text variable: DALI_Commissioning.fbPart102Scenes.aScene[19], input disabled if: DALI_Commissioning.fbPart102Scenes.aNoShortAddress[19]
                p55702900: DALI_Commissioning.fbPart102Scenes.aFont[19]
                OnMouseClick: write the text variable via Default, min 0, max 255, title "Scene Value"
        Group (295,120 65x30)
            Textfield (0,0 30x30), "20"
            Textfield (30,0 35x30), "%s", text variable: DALI_Commissioning.fbPart102Scenes.aScene[20], input disabled if: DALI_Commissioning.fbPart102Scenes.aNoShortAddress[20]
                p55702900: DALI_Commissioning.fbPart102Scenes.aFont[20]
                OnMouseClick: write the text variable via Default, min 0, max 255, title "Scene Value"
        Group (365,120 65x30)
            Textfield (0,0 30x30), "21"
            Textfield (30,0 35x30), "%s", text variable: DALI_Commissioning.fbPart102Scenes.aScene[21], input disabled if: DALI_Commissioning.fbPart102Scenes.aNoShortAddress[21]
                p55702900: DALI_Commissioning.fbPart102Scenes.aFont[21]
                OnMouseClick: write the text variable via Default, min 0, max 255, title "Scene Value"
        Group (435,120 65x30)
            Textfield (0,0 30x30), "22"
            Textfield (30,0 35x30), "%s", text variable: DALI_Commissioning.fbPart102Scenes.aScene[22], input disabled if: DALI_Commissioning.fbPart102Scenes.aNoShortAddress[22]
                p55702900: DALI_Commissioning.fbPart102Scenes.aFont[22]
                OnMouseClick: write the text variable via Default, min 0, max 255, title "Scene Value"
        Group (505,120 65x30)
            Textfield (0,0 30x30), "23"
            Textfield (30,0 35x30), "%s", text variable: DALI_Commissioning.fbPart102Scenes.aScene[23], input disabled if: DALI_Commissioning.fbPart102Scenes.aNoShortAddress[23]
                p55702900: DALI_Commissioning.fbPart102Scenes.aFont[23]
                OnMouseClick: write the text variable via Default, min 0, max 255, title "Scene Value"
        Group (85,165 65x30)
            Textfield (0,0 30x30), "25"
            Textfield (30,0 35x30), "%s", text variable: DALI_Commissioning.fbPart102Scenes.aScene[25], input disabled if: DALI_Commissioning.fbPart102Scenes.aNoShortAddress[25]
                p55702900: DALI_Commissioning.fbPart102Scenes.aFont[25]
                OnMouseClick: write the text variable via Default, min 0, max 255, title "Scene Value"
        Group (155,165 65x30)
            Textfield (0,0 30x30), "26"
            Textfield (30,0 35x30), "%s", text variable: DALI_Commissioning.fbPart102Scenes.aScene[26], input disabled if: DALI_Commissioning.fbPart102Scenes.aNoShortAddress[26]
                p55702900: DALI_Commissioning.fbPart102Scenes.aFont[26]
                OnMouseClick: write the text variable via Default, min 0, max 255, title "Scene Value"
        Group (225,165 65x30)
            Textfield (0,0 30x30), "27"
            Textfield (30,0 35x30), "%s", text variable: DALI_Commissioning.fbPart102Scenes.aScene[27], input disabled if: DALI_Commissioning.fbPart102Scenes.aNoShortAddress[27]
                p55702900: DALI_Commissioning.fbPart102Scenes.aFont[27]
                OnMouseClick: write the text variable via Default, min 0, max 255, title "Scene Value"
        Group (295,165 65x30)
            Textfield (0,0 30x30), "28"
            Textfield (30,0 35x30), "%s", text variable: DALI_Commissioning.fbPart102Scenes.aScene[28], input disabled if: DALI_Commissioning.fbPart102Scenes.aNoShortAddress[28]
                p55702900: DALI_Commissioning.fbPart102Scenes.aFont[28]
                OnMouseClick: write the text variable via Default, min 0, max 255, title "Scene Value"
        Group (365,165 65x30)
            Textfield (0,0 30x30), "29"
            Textfield (30,0 35x30), "%s", text variable: DALI_Commissioning.fbPart102Scenes.aScene[29], input disabled if: DALI_Commissioning.fbPart102Scenes.aNoShortAddress[29]
                p55702900: DALI_Commissioning.fbPart102Scenes.aFont[29]
                OnMouseClick: write the text variable via Default, min 0, max 255, title "Scene Value"
        Group (435,165 65x30)
            Textfield (0,0 30x30), "30"
            Textfield (30,0 35x30), "%s", text variable: DALI_Commissioning.fbPart102Scenes.aScene[30], input disabled if: DALI_Commissioning.fbPart102Scenes.aNoShortAddress[30]
                p55702900: DALI_Commissioning.fbPart102Scenes.aFont[30]
                OnMouseClick: write the text variable via Default, min 0, max 255, title "Scene Value"
        Group (505,165 65x30)
            Textfield (0,0 30x30), "31"
            Textfield (30,0 35x30), "%s", text variable: DALI_Commissioning.fbPart102Scenes.aScene[31], input disabled if: DALI_Commissioning.fbPart102Scenes.aNoShortAddress[31]
                p55702900: DALI_Commissioning.fbPart102Scenes.aFont[31]
                OnMouseClick: write the text variable via Default, min 0, max 255, title "Scene Value"
        Group (85,210 65x30)
            Textfield (0,0 30x30), "33"
            Textfield (30,0 35x30), "%s", text variable: DALI_Commissioning.fbPart102Scenes.aScene[33], input disabled if: DALI_Commissioning.fbPart102Scenes.aNoShortAddress[32]
                p55702900: DALI_Commissioning.fbPart102Scenes.aFont[33]
                OnMouseClick: write the text variable via Default, min 0, max 255, title "Scene Value"
        Group (155,210 65x30)
            Textfield (0,0 30x30), "34"
            Textfield (30,0 35x30), "%s", text variable: DALI_Commissioning.fbPart102Scenes.aScene[34], input disabled if: DALI_Commissioning.fbPart102Scenes.aNoShortAddress[34]
                p55702900: DALI_Commissioning.fbPart102Scenes.aFont[34]
                OnMouseClick: write the text variable via Default, min 0, max 255, title "Scene Value"
        Group (295,210 65x30)
            Textfield (0,0 30x30), "36"
            Textfield (30,0 35x30), "%s", text variable: DALI_Commissioning.fbPart102Scenes.aScene[36], input disabled if: DALI_Commissioning.fbPart102Scenes.aNoShortAddress[36]
                p55702900: DALI_Commissioning.fbPart102Scenes.aFont[36]
                OnMouseClick: write the text variable via Default, min 0, max 255
        Group (365,210 65x30)
            Textfield (0,0 30x30), "37"
            Textfield (30,0 35x30), "%s", text variable: DALI_Commissioning.fbPart102Scenes.aScene[37], input disabled if: DALI_Commissioning.fbPart102Scenes.aNoShortAddress[37]
                p55702900: DALI_Commissioning.fbPart102Scenes.aFont[37]
                OnMouseClick: write the text variable via Default, min 0, max 255, title "Scene Value"
        Group (435,210 65x30)
            Textfield (0,0 30x30), "38"
            Textfield (30,0 35x30), "%s", text variable: DALI_Commissioning.fbPart102Scenes.aScene[38], input disabled if: DALI_Commissioning.fbPart102Scenes.aNoShortAddress[38]
                p55702900: DALI_Commissioning.fbPart102Scenes.aFont[38]
                OnMouseClick: write the text variable via Default, min 0, max 255, title "Scene Value"
        Group (505,210 65x30)
            Textfield (0,0 30x30), "39"
            Textfield (30,0 35x30), "%s", text variable: DALI_Commissioning.fbPart102Scenes.aScene[39], input disabled if: DALI_Commissioning.fbPart102Scenes.aNoShortAddress[39]
                p55702900: DALI_Commissioning.fbPart102Scenes.aFont[39]
                OnMouseClick: write the text variable via Default, min 0, max 255, title "Scene Value"
        Group (85,255 65x30)
            Textfield (0,0 30x30), "41"
            Textfield (30,0 35x30), "%s", text variable: DALI_Commissioning.fbPart102Scenes.aScene[41], input disabled if: DALI_Commissioning.fbPart102Scenes.aNoShortAddress[41]
                p55702900: DALI_Commissioning.fbPart102Scenes.aFont[41]
                OnMouseClick: write the text variable via Default, min 0, max 255, title "Scene Value"
        Group (155,255 65x30)
            Textfield (0,0 30x30), "42"
            Textfield (30,0 35x30), "%s", text variable: DALI_Commissioning.fbPart102Scenes.aScene[42], input disabled if: DALI_Commissioning.fbPart102Scenes.aNoShortAddress[42]
                p55702900: DALI_Commissioning.fbPart102Scenes.aFont[42]
                OnMouseClick: write the text variable via Default, min 0, max 255, title "Scene Value"
        Group (225,210 65x30)
            Textfield (0,0 30x30), "35"
            Textfield (30,0 35x30), "%s", text variable: DALI_Commissioning.fbPart102Scenes.aScene[35], input disabled if: DALI_Commissioning.fbPart102Scenes.aNoShortAddress[35]
                p55702900: DALI_Commissioning.fbPart102Scenes.aFont[35]
                OnMouseClick: write the text variable via Default, min 0, max 255, title "Scene Value"
        Group (225,255 65x30)
            Textfield (0,0 30x30), "43"
            Textfield (30,0 35x30), "%s", text variable: DALI_Commissioning.fbPart102Scenes.aScene[43], input disabled if: DALI_Commissioning.fbPart102Scenes.aNoShortAddress[43]
                p55702900: DALI_Commissioning.fbPart102Scenes.aFont[43]
                OnMouseClick: write the text variable via Default, min 0, max 255, title "Scene Value"
        Group (295,255 65x30)
            Textfield (0,0 30x30), "44"
            Textfield (30,0 35x30), "%s", text variable: DALI_Commissioning.fbPart102Scenes.aScene[44], input disabled if: DALI_Commissioning.fbPart102Scenes.aNoShortAddress[44]
                p55702900: DALI_Commissioning.fbPart102Scenes.aFont[44]
                OnMouseClick: write the text variable via Default, min 0, max 255, title "Scene Value"
        Group (365,255 65x30)
            Textfield (0,0 30x30), "45"
            Textfield (30,0 35x30), "%s", text variable: DALI_Commissioning.fbPart102Scenes.aScene[45], input disabled if: DALI_Commissioning.fbPart102Scenes.aNoShortAddress[45]
                p55702900: DALI_Commissioning.fbPart102Scenes.aFont[45]
                OnMouseClick: write the text variable via Default, min 0, max 255, title "Scene Value"
        Group (435,255 65x30)
            Textfield (0,0 30x30), "46"
            Textfield (30,0 35x30), "%s", text variable: DALI_Commissioning.fbPart102Scenes.aScene[46], input disabled if: DALI_Commissioning.fbPart102Scenes.aNoShortAddress[46]
                p55702900: DALI_Commissioning.fbPart102Scenes.aFont[46]
                OnMouseClick: write the text variable via Default, min 0, max 255, title "Scene Value"
        Group (505,255 65x30)
            Textfield (0,0 30x30), "47"
            Textfield (30,0 35x30), "%s", text variable: DALI_Commissioning.fbPart102Scenes.aScene[47], input disabled if: DALI_Commissioning.fbPart102Scenes.aNoShortAddress[47]
                p55702900: DALI_Commissioning.fbPart102Scenes.aFont[47]
                OnMouseClick: write the text variable via Default, min 0, max 255, title "Scene Value"
        Group (85,300 65x30)
            Textfield (0,0 30x30), "49"
            Textfield (30,0 35x30), "%s", text variable: DALI_Commissioning.fbPart102Scenes.aScene[49], input disabled if: DALI_Commissioning.fbPart102Scenes.aNoShortAddress[49]
                p55702900: DALI_Commissioning.fbPart102Scenes.aFont[49]
                OnMouseClick: write the text variable via Default, min 0, max 255, title "Scene Value"
        Group (155,300 65x30)
            Textfield (0,0 30x30), "50"
            Textfield (30,0 35x30), "%s", text variable: DALI_Commissioning.fbPart102Scenes.aScene[50], input disabled if: DALI_Commissioning.fbPart102Scenes.aNoShortAddress[50]
                p55702900: DALI_Commissioning.fbPart102Scenes.aFont[50]
                OnMouseClick: write the text variable via Default, min 0, max 255, title "Scene Value"
        Group (225,300 65x30)
            Textfield (0,0 30x30), "51"
            Textfield (30,0 35x30), "%s", text variable: DALI_Commissioning.fbPart102Scenes.aScene[51], input disabled if: DALI_Commissioning.fbPart102Scenes.aNoShortAddress[51]
                p55702900: DALI_Commissioning.fbPart102Scenes.aFont[51]
                OnMouseClick: write the text variable via Default, min 0, max 255, title "Scene Value"
        Group (295,300 65x30)
            Textfield (0,0 30x30), "52"
            Textfield (30,0 35x30), "%s", text variable: DALI_Commissioning.fbPart102Scenes.aScene[52], input disabled if: DALI_Commissioning.fbPart102Scenes.aNoShortAddress[52]
                p55702900: DALI_Commissioning.fbPart102Scenes.aFont[52]
                OnMouseClick: write the text variable via Default, min 0, max 255, title "Scene Value"
        Group (365,300 65x30)
            Textfield (0,0 30x30), "53"
            Textfield (30,0 35x30), "%s", text variable: DALI_Commissioning.fbPart102Scenes.aScene[53], input disabled if: DALI_Commissioning.fbPart102Scenes.aNoShortAddress[53]
                p55702900: DALI_Commissioning.fbPart102Scenes.aFont[53]
                OnMouseClick: write the text variable via Default, min 0, max 255, title "Scene Value"
        Group (435,300 64x30)
            Textfield (0,0 29x30), "54"
            Textfield (29,0 35x30), "%s", text variable: DALI_Commissioning.fbPart102Scenes.aScene[54], input disabled if: DALI_Commissioning.fbPart102Scenes.aNoShortAddress[54]
                p55702900: DALI_Commissioning.fbPart102Scenes.aFont[54]
                OnMouseClick: write the text variable via Default, min 0, max 255, title "Scene Value"
        Group (505,300 65x30)
            Textfield (0,0 30x30), "55"
            Textfield (30,0 35x30), "%s", text variable: DALI_Commissioning.fbPart102Scenes.aScene[55], input disabled if: DALI_Commissioning.fbPart102Scenes.aNoShortAddress[55]
                p55702900: DALI_Commissioning.fbPart102Scenes.aFont[55]
                OnMouseClick: write the text variable via Default, min 0, max 255, title "Scene Value"
        Group (85,345 65x30)
            Textfield (0,0 30x30), "57"
            Textfield (30,0 35x30), "%s", text variable: DALI_Commissioning.fbPart102Scenes.aScene[57], input disabled if: DALI_Commissioning.fbPart102Scenes.aNoShortAddress[57]
                p55702900: DALI_Commissioning.fbPart102Scenes.aFont[57]
                OnMouseClick: write the text variable via Default, min 0, max 255, title "Scene Value"
        Group (155,345 65x30)
            Textfield (0,0 30x30), "58"
            Textfield (30,0 35x30), "%s", text variable: DALI_Commissioning.fbPart102Scenes.aScene[58], input disabled if: DALI_Commissioning.fbPart102Scenes.aNoShortAddress[58]
                p55702900: DALI_Commissioning.fbPart102Scenes.aFont[58]
                OnMouseClick: write the text variable via Default, min 0, max 255, title "Scene Value"
        Group (225,345 65x30)
            Textfield (0,0 30x30), "59"
            Textfield (30,0 35x30), "%s", text variable: DALI_Commissioning.fbPart102Scenes.aScene[59], input disabled if: DALI_Commissioning.fbPart102Scenes.aNoShortAddress[59]
                p55702900: DALI_Commissioning.fbPart102Scenes.aFont[59]
                OnMouseClick: write the text variable via Default, min 0, max 255, title "Scene Value"
        Group (295,345 65x30)
            Textfield (0,0 30x30), "60"
            Textfield (30,0 35x30), "%s", text variable: DALI_Commissioning.fbPart102Scenes.aScene[60], input disabled if: DALI_Commissioning.fbPart102Scenes.aNoShortAddress[60]
                p55702900: DALI_Commissioning.fbPart102Scenes.aFont[60]
                OnMouseClick: write the text variable via Default, min 0, max 255, title "Scene Value"
        Group (365,345 65x30)
            Textfield (0,0 30x30), "61"
            Textfield (30,0 35x30), "%s", text variable: DALI_Commissioning.fbPart102Scenes.aScene[61], input disabled if: DALI_Commissioning.fbPart102Scenes.aNoShortAddress[61]
                p55702900: DALI_Commissioning.fbPart102Scenes.aFont[61]
                OnMouseClick: write the text variable via Default, min 0, max 255, title "Scene Value"
        Group (435,345 65x30)
            Textfield (0,0 30x30), "62"
            Textfield (30,0 35x30), "%s", text variable: DALI_Commissioning.fbPart102Scenes.aScene[62], input disabled if: DALI_Commissioning.fbPart102Scenes.aNoShortAddress[62]
                p55702900: DALI_Commissioning.fbPart102Scenes.aFont[62]
                OnMouseClick: write the text variable via Default, min 0, max 255, title "Scene Value"
        Group (505,345 65x30)
            Textfield (0,0 30x30), "63"
            Textfield (30,0 35x30), "%s", text variable: DALI_Commissioning.fbPart102Scenes.aScene[63], input disabled if: DALI_Commissioning.fbPart102Scenes.aNoShortAddress[63]
                p55702900: DALI_Commissioning.fbPart102Scenes.aFont[63]
                OnMouseClick: write the text variable via Default, min 0, max 255, title "Scene Value"
        WaitingSymbolFlower (240,170 70x70), invisible if: DALI_Commissioning.fbPart102Scenes.bHideWaitSymbol
        Group (15,30 65x30)
            Textfield (0,0 30x30), "0"
            Textfield (30,0 35x30), "%s", text variable: DALI_Commissioning.fbPart102Scenes.aScene[0], input disabled if: DALI_Commissioning.fbPart102Scenes.aNoShortAddress[0]
                p55702900: DALI_Commissioning.fbPart102Scenes.aFont[0]
                OnMouseClick: write the text variable via Default, min 0, max 255, title "Scene Value"
    Button (620,400 150x40), "Read"
        OnMouseClick: execute { DALI_Commissioning.fbPart102Scenes.bRead := TRUE; }
    Button (620,450 150x40), "Write"
        OnMouseClick: execute { DALI_Commissioning.fbPart102Scenes.bWrite := TRUE; }
    Button (620,100 150x40), "Go to scene"
        OnMouseClick: execute { DALI_Commissioning.fbPart102Scenes.bGoToScene := TRUE; }
    Button (620,150 150x40), "Switch Off"
        OnMouseClick: execute { DALI_Commissioning.fbPart102Scenes.bSwitchOff := TRUE; }
    Textfield (390,10 120x40), "Choose scene:"
    Button (520,10 80x40), "%s", text variable: DALI_Commissioning.fbPart102Scenes.nScene
        OnMouseClick: write the text variable via Default, min 0, max 15, title "Choose scene"
    Group (10,5 170x40)
        Textfield (0,0 110x40), "DALI Line:"
        Button (90,0 80x40), "%d", text variable: GVL_Internal.nDALILine
            OnMouseClick: write the text variable via Default, min 1, max 10, title "Choose line"
END_VISUALIZATION

